C03576=1018.890,246.448,-130.544,169.177,50.795,159.695
C03577=1018.883,246.200,-130.516,169.173,50.800,159.695
C03578=1018.878,245.952,-130.488,169.170,50.806,159.696
C03579=1018.872,245.703,-130.460,169.165,50.812,159.696
C03580=1018.866,245.455,-130.433,169.160,50.817,159.697
C03581=1018.860,245.206,-130.405,169.156,50.823,159.697
C03582=1018.855,244.958,-130.377,169.152,50.829,159.698
C03583=1018.848,244.709,-130.349,169.148,50.834,159.698
C03584=1018.843,244.461,-130.321,169.143,50.840,159.699
C03585=1018.836,244.213,-130.294,169.139,50.846,159.699
C03586=1018.831,243.964,-130.266,169.135,50.852,159.700
C03587=1018.825,243.715,-130.238,169.131,50.857,159.700
C03588=1018.819,243.468,-130.211,169.126,50.863,159.701
C03589=1018.813,243.219,-130.182,169.122,50.869,159.701
C03590=1018.807,242.971,-130.156,169.118,50.875,159.702
C03591=1018.802,242.723,-130.128,169.113,50.881,159.702
C03592=1018.795,242.473,-130.101,169.109,50.887,159.703
C03593=1018.789,242.226,-130.073,169.104,50.893,159.703
C03594=1018.784,241.976,-130.046,169.101,50.899,159.704
C03595=1018.778,241.729,-130.018,169.095,50.904,159.704
C03596=1018.771,241.480,-129.991,169.092,50.910,159.705
C03597=1018.766,241.232,-129.963,169.088,50.917,159.706
C03598=1018.760,240.983,-129.937,169.083,50.922,159.706
C03599=1018.753,240.735,-129.909,169.079,50.928,159.707
C03600=1018.748,240.486,-129.882,169.074,50.934,159.707
C03601=1018.742,240.238,-129.854,169.071,50.940,159.708
C03602=1018.736,239.989,-129.827,169.067,50.946,159.709
C03603=1018.731,239.741,-129.799,169.062,50.952,159.709
C03604=1018.724,239.492,-129.772,169.058,50.958,159.710
C03605=1018.718,239.244,-129.745,169.053,50.965,159.710
C03606=1018.713,238.996,-129.718,169.049,50.970,159.711
C03607=1018.707,238.747,-129.691,169.045,50.976,159.711
C03608=1018.701,238.499,-129.663,169.041,50.983,159.712
C03609=1018.694,238.250,-129.636,169.036,50.989,159.712
C03610=1018.688,238.002,-129.610,169.033,50.995,159.713
C03611=1018.683,237.753,-129.583,169.028,51.001,159.714
C03612=1018.676,237.505,-129.555,169.024,51.007,159.714
C03613=1018.670,237.256,-129.529,169.019,51.013,159.715
C03614=1018.664,237.008,-129.502,169.016,51.020,159.715
C03615=1018.658,236.759,-129.475,169.011,51.026,159.716
C03616=1018.652,236.511,-129.448,169.007,51.032,159.717
C03617=1018.646,236.263,-129.421,169.004,51.038,159.717
C03618=1018.641,236.013,-129.393,168.999,51.045,159.718
C03619=1018.635,235.765,-129.367,168.994,51.051,159.719
C03620=1018.629,235.517,-129.340,168.991,51.057,159.719
C03621=1018.623,235.268,-129.313,168.985,51.063,159.720
C03622=1018.617,235.019,-129.286,168.982,51.069,159.720
C03623=1018.611,234.792,-129.262,168.978,51.075,159.721
C03624=1018.605,234.565,-129.237,168.974,51.081,159.721
C03625=1018.600,234.338,-129.213,168.970,51.087,159.722
C03626=1018.595,234.111,-129.189,168.966,51.092,159.723
C03627=1018.590,233.885,-129.164,168.963,51.098,159.723
C03628=1018.584,233.657,-129.140,168.959,51.104,159.724
C03629=1018.578,233.430,-129.115,168.955,51.110,159.724
C03630=1018.573,233.203,-129.090,168.951,51.116,159.725
C03631=1018.567,232.954,-129.064,168.948,51.122,159.726
C03632=1018.562,232.706,-129.037,168.943,51.129,159.726
C03633=1018.555,232.457,-129.010,168.939,51.135,159.727
C03634=1018.550,232.209,-128.983,168.935,51.141,159.728
C03635=1018.544,231.960,-128.957,168.931,51.147,159.728
C03636=1018.538,231.712,-128.930,168.926,51.154,159.729
C03637=1018.532,231.464,-128.903,168.922,51.160,159.729
C03638=1018.526,231.214,-128.877,168.918,51.166,159.730
C03639=1018.520,230.966,-128.850,168.913,51.173,159.731
C03640=1018.515,230.717,-128.824,168.910,51.180,159.731
C03641=1018.509,230.469,-128.797,168.906,51.186,159.732
C03642=1018.503,230.220,-128.770,168.902,51.192,159.733
C03643=1018.497,229.972,-128.744,168.897,51.199,159.733
C03644=1018.490,229.723,-128.717,168.894,51.205,159.734
C03645=1018.484,229.475,-128.691,168.889,51.212,159.735
C03646=1018.479,229.226,-128.665,168.885,51.218,159.735
C03647=1018.473,228.978,-128.638,168.881,51.225,159.736
C03648=1018.467,228.729,-128.611,168.877,51.232,159.737
C03649=1018.462,228.481,-128.585,168.873,51.238,159.737
C03650=1018.455,228.233,-128.559,168.868,51.244,159.738
C03651=1018.450,227.984,-128.533,168.864,51.252,159.739
C03652=1018.443,227.735,-128.506,168.861,51.258,159.739
C03653=1018.437,227.486,-128.479,168.856,51.264,159.740
C03654=1018.432,227.238,-128.453,168.853,51.271,159.741
C03655=1018.426,226.989,-128.427,168.848,51.278,159.742
C03656=1018.420,226.741,-128.401,168.843,51.284,159.742
C03657=1018.414,226.493,-128.374,168.840,51.291,159.743
C03658=1018.409,226.244,-128.348,168.836,51.297,159.744
C03659=1018.402,225.996,-128.322,168.832,51.304,159.744
C03660=1018.397,225.747,-128.296,168.828,51.311,159.745
C03661=1018.391,225.498,-128.269,168.823,51.318,159.746
C03662=1018.385,225.250,-128.244,168.819,51.324,159.746
C03663=1018.379,225.001,-128.217,168.816,51.331,159.747
C03664=1018.372,224.752,-128.192,168.811,51.338,159.748
C03665=1018.366,224.504,-128.165,168.807,51.345,159.749
C03666=1018.360,224.255,-128.140,168.804,51.352,159.749
C03667=1018.354,224.007,-128.113,168.799,51.358,159.750
C03668=1018.349,223.758,-128.087,168.795,51.365,159.751
C03669=1018.342,223.510,-128.061,168.791,51.372,159.752
C03670=1018.337,223.261,-128.035,168.787,51.379,159.752
C03671=1018.330,223.013,-128.009,168.783,51.386,159.753
C03672=1018.325,222.764,-127.983,168.779,51.393,159.754
C03673=1018.319,222.515,-127.957,168.775,51.399,159.755
C03674=1018.313,222.267,-127.931,168.770,51.406,159.755
C03675=1018.307,222.018,-127.905,168.766,51.414,159.756
C03676=1018.301,221.769,-127.879,168.763,51.420,159.757
C03677=1018.295,221.521,-127.853,168.758,51.427,159.758
C03678=1018.289,221.272,-127.828,168.754,51.434,159.758
C03679=1018.283,221.023,-127.801,168.751,51.440,159.759
C03680=1018.278,220.774,-127.775,168.746,51.448,159.760
C03681=1018.272,220.526,-127.750,168.742,51.455,159.761
C03682=1018.266,220.277,-127.723,168.738,51.462,159.761
C03683=1018.261,220.047,-127.699,168.734,51.468,159.762
C03684=1018.255,219.815,-127.676,168.731,51.474,159.763
C03685=1018.250,219.583,-127.651,168.728,51.481,159.764
C03686=1018.244,219.353,-127.628,168.723,51.488,159.764
C03687=1018.239,219.122,-127.603,168.719,51.494,159.765
C03688=1018.234,218.890,-127.579,168.716,51.501,159.766
C03689=1018.228,218.659,-127.556,168.713,51.507,159.766
C03690=1018.222,218.428,-127.531,168.708,51.513,159.767
C03691=1018.217,218.179,-127.505,168.705,51.520,159.768
C03692=1018.211,217.930,-127.480,168.701,51.527,159.769
C03693=1018.205,217.682,-127.455,168.696,51.535,159.769
C03694=1018.200,217.433,-127.429,168.692,51.542,159.770
C03695=1018.193,217.185,-127.403,168.688,51.549,159.771
C03696=1018.187,216.936,-127.378,168.685,51.556,159.772
C03697=1018.181,216.687,-127.352,168.681,51.563,159.773
C03698=1018.175,216.439,-127.327,168.676,51.570,159.773
C03699=1018.169,216.190,-127.301,168.672,51.578,159.774
C03700=1018.163,215.941,-127.276,168.668,51.585,159.775
C03701=1018.158,215.693,-127.250,168.664,51.592,159.776
C03702=1018.152,215.444,-127.225,168.661,51.599,159.777
C03703=1018.146,215.196,-127.200,168.657,51.607,159.778
C03704=1018.140,214.947,-127.174,168.653,51.614,159.778
C03705=1018.134,214.698,-127.148,168.648,51.621,159.779
C03706=1018.128,214.450,-127.123,168.644,51.629,159.780
C03707=1018.122,214.202,-127.098,168.640,51.636,159.781
C03708=1018.117,213.953,-127.072,168.637,51.643,159.782
C03709=1018.110,213.704,-127.047,168.633,51.650,159.782
C03710=1018.104,213.455,-127.021,168.629,51.658,159.783
C03711=1018.098,213.207,-126.996,168.625,51.665,159.784
C03712=1018.093,212.958,-126.971,168.621,51.672,159.785
C03713=1018.087,212.709,-126.946,168.616,51.680,159.786
C03714=1018.081,212.460,-126.921,168.612,51.687,159.787
C03715=1018.076,212.211,-126.895,168.609,51.694,159.787
C03716=1018.069,211.963,-126.869,168.605,51.702,159.788
C03717=1018.064,211.715,-126.844,168.601,51.709,159.789
C03718=1018.058,211.466,-126.819,168.597,51.716,159.790
C03719=1018.052,211.217,-126.793,168.593,51.723,159.791
C03720=1018.046,210.968,-126.768,168.589,51.731,159.792
C03721=1018.041,210.720,-126.743,168.585,51.739,159.793
C03722=1018.034,210.471,-126.718,168.581,51.746,159.793
C03723=1018.029,210.222,-126.692,168.578,51.753,159.794
C03724=1018.023,209.974,-126.667,168.574,51.761,159.795
C03725=1018.017,209.726,-126.642,168.570,51.768,159.796
C03726=1018.011,209.476,-126.617,168.566,51.776,159.797
C03727=1018.006,209.228,-126.592,168.562,51.783,159.798
C03728=1017.999,208.980,-126.567,168.557,51.790,159.799
C03729=1017.993,208.730,-126.542,168.554,51.798,159.800
C03730=1017.988,208.481,-126.516,168.550,51.806,159.800
C03731=1017.982,208.233,-126.491,168.546,51.813,159.801
C03732=1017.976,207.984,-126.467,168.542,51.821,159.802
C03733=1017.970,207.735,-126.441,168.538,51.829,159.803
C03734=1017.965,207.487,-126.417,168.534,51.836,159.804
C03735=1017.959,207.238,-126.392,168.530,51.844,159.805
C03736=1017.953,206.989,-126.367,168.526,51.851,159.806
C03737=1017.947,206.741,-126.342,168.522,51.859,159.807
C03738=1017.941,206.492,-126.317,168.518,51.866,159.807
C03739=1017.935,206.244,-126.292,168.514,51.874,159.808
C03740=1017.930,205.995,-126.267,168.511,51.882,159.809
C03741=1017.923,205.746,-126.242,168.506,51.890,159.810
C03742=1017.918,205.498,-126.218,168.503,51.898,159.811
C03743=1017.912,205.264,-126.195,168.500,51.904,159.812
C03744=1017.907,205.031,-126.171,168.495,51.912,159.813
C03745=1017.901,204.798,-126.148,168.491,51.919,159.814
C03746=1017.895,204.565,-126.125,168.489,51.927,159.815
C03747=1017.890,204.332,-126.102,168.484,51.934,159.816
C03748=1017.885,204.098,-126.078,168.481,51.941,159.816
C03749=1017.879,203.865,-126.055,168.478,51.949,159.817
C03750=1017.854,202.631,-125.940,167.998,51.859,159.707
C03751=1017.849,202.382,-125.916,167.994,51.868,159.708
C03752=1017.844,202.134,-125.893,167.989,51.876,159.709
C03753=1017.839,201.884,-125.870,167.984,51.885,159.710
C03754=1017.834,201.636,-125.847,167.980,51.894,159.711
C03755=1017.828,201.387,-125.824,167.976,51.903,159.712
C03756=1017.824,201.138,-125.801,167.971,51.912,159.713
C03757=1017.819,200.889,-125.778,167.966,51.921,159.714
C03758=1017.815,200.640,-125.755,167.962,51.930,159.715
C03759=1017.809,200.391,-125.732,167.956,51.938,159.716
C03760=1017.805,200.143,-125.709,167.952,51.947,159.717
C03761=1017.800,199.893,-125.686,167.948,51.956,159.718
C03762=1017.795,199.645,-125.663,167.943,51.965,159.719
C03763=1017.790,199.395,-125.640,167.938,51.974,159.720
C03764=1017.785,199.147,-125.617,167.934,51.983,159.721
C03765=1017.780,198.897,-125.594,167.930,51.992,159.722
C03766=1017.775,198.649,-125.572,167.925,52.001,159.723
C03767=1017.770,198.400,-125.549,167.921,52.010,159.724
C03768=1017.765,198.151,-125.526,167.916,52.019,159.725
C03769=1017.760,197.902,-125.504,167.912,52.028,159.726
C03770=1017.755,197.654,-125.481,167.907,52.037,159.727
C03771=1017.750,197.404,-125.459,167.903,52.046,159.728
C03772=1017.745,197.156,-125.436,167.898,52.055,159.729
C03773=1017.739,196.906,-125.414,167.893,52.064,159.730
C03774=1017.735,196.657,-125.391,167.889,52.073,159.731
C03775=1017.730,196.408,-125.368,167.885,52.082,159.732
C03776=1017.725,196.159,-125.346,167.880,52.091,159.733
C03777=1017.720,195.911,-125.323,167.875,52.100,159.734
C03778=1017.715,195.661,-125.301,167.871,52.109,159.735
C03779=1017.710,195.413,-125.278,167.867,52.118,159.736
C03780=1017.704,195.163,-125.256,167.862,52.127,159.737
C03781=1017.700,194.915,-125.233,167.858,52.136,159.738
C03782=1017.695,194.666,-125.211,167.854,52.145,159.739
C03783=1017.690,194.417,-125.189,167.849,52.154,159.740
C03784=1017.685,194.168,-125.166,167.845,52.163,159.741
C03785=1017.681,193.919,-125.144,167.841,52.173,159.742
C03786=1017.675,193.670,-125.122,167.836,52.182,159.743
C03787=1017.671,193.421,-125.099,167.832,52.191,159.744
C03788=1017.666,193.172,-125.077,167.827,52.199,159.745
C03789=1017.661,192.923,-125.054,167.823,52.208,159.746
C03790=1017.656,192.674,-125.031,167.819,52.217,159.747
C03791=1017.651,192.426,-125.009,167.814,52.226,159.748
C03792=1017.646,192.176,-124.987,167.810,52.236,159.749
C03793=1017.641,191.927,-124.965,167.806,52.245,159.750
C03794=1017.637,191.679,-124.942,167.801,52.254,159.751
C03795=1017.631,191.429,-124.920,167.797,52.263,159.752
C03796=1017.626,191.180,-124.898,167.793,52.272,159.753
C03797=1017.622,190.931,-124.876,167.788,52.281,159.754
C03798=1017.617,190.683,-124.853,167.784,52.290,159.755
C03799=1017.612,190.434,-124.831,167.780,52.299,159.756
C03800=1017.607,190.185,-124.809,167.775,52.308,159.757
C03801=1017.603,189.936,-124.786,167.771,52.317,159.758
C03802=1017.598,189.687,-124.765,167.766,52.326,159.759
C03803=1017.592,189.438,-124.742,167.762,52.335,159.760
C03804=1017.588,189.189,-124.719,167.758,52.344,159.761
C03805=1017.583,188.940,-124.697,167.754,52.353,159.762
C03806=1017.579,188.691,-124.675,167.750,52.362,159.764
C03807=1017.574,188.441,-124.653,167.746,52.371,159.765
C03808=1017.569,188.193,-124.631,167.742,52.381,159.766
C03809=1017.564,187.944,-124.609,167.737,52.390,159.767
C03810=1017.559,187.696,-124.586,167.733,52.399,159.768
C03811=1017.554,187.415,-124.561,167.728,52.409,159.769
C03812=1017.548,187.135,-124.536,167.723,52.419,159.770
C03813=1017.544,186.854,-124.511,167.719,52.429,159.771
C03814=1017.538,186.573,-124.486,167.714,52.440,159.772
C03815=1017.534,186.324,-124.464,167.710,52.448,159.773
C03816=1017.529,186.076,-124.442,167.706,52.458,159.774
C03817=1017.524,185.826,-124.420,167.702,52.467,159.775
C03818=1017.519,185.577,-124.398,167.698,52.476,159.777
C03819=1017.515,185.328,-124.375,167.693,52.485,159.778
C03820=1017.510,185.079,-124.354,167.689,52.493,159.778
C03821=1017.505,184.830,-124.332,167.685,52.502,159.780
C03822=1017.500,184.582,-124.310,167.681,52.511,159.781
C03823=1017.496,184.333,-124.287,167.677,52.521,159.782
C03824=1017.491,184.084,-124.266,167.673,52.530,159.783
C03825=1017.486,183.835,-124.244,167.668,52.539,159.784
C03826=1017.482,183.586,-124.221,167.664,52.548,159.785
C03827=1017.477,183.336,-124.199,167.661,52.557,159.786
C03828=1017.472,183.087,-124.178,167.657,52.566,159.787
C03829=1017.468,182.838,-124.156,167.652,52.575,159.788
C03830=1017.463,182.589,-124.134,167.648,52.584,159.789
C03831=1017.459,182.340,-124.112,167.644,52.594,159.790
C03832=1017.454,182.091,-124.090,167.641,52.602,159.791
C03833=1017.450,181.842,-124.067,167.636,52.611,159.792
C03834=1017.444,181.593,-124.047,167.632,52.621,159.793
C03835=1017.440,181.344,-124.025,167.628,52.630,159.794
C03836=1017.435,181.095,-124.004,167.624,52.639,159.795
C03837=1017.429,180.846,-123.982,167.619,52.648,159.796
C03838=1017.424,180.597,-123.960,167.616,52.658,159.798
C03839=1017.419,180.348,-123.940,167.611,52.667,159.799
C03840=1017.414,180.099,-123.918,167.607,52.677,159.800
C03841=1017.410,179.849,-123.897,167.603,52.687,159.801
C03842=1017.404,179.601,-123.875,167.599,52.696,159.802
C03843=1017.399,179.351,-123.854,167.595,52.705,159.803
C03844=1017.395,179.103,-123.832,167.591,52.714,159.804
C03845=1017.389,178.853,-123.812,167.587,52.724,159.805
C03846=1017.385,178.605,-123.790,167.583,52.733,159.806
C03847=1017.380,178.355,-123.769,167.579,52.742,159.808
C03848=1017.374,178.107,-123.748,167.575,52.751,159.809
C03849=1017.370,177.857,-123.726,167.571,52.761,159.810
C03850=1017.365,177.608,-123.706,167.567,52.770,159.811
C03851=1017.360,177.359,-123.684,167.563,52.780,159.812
C03852=1017.355,177.110,-123.663,167.559,52.789,159.813
C03853=1017.350,176.861,-123.642,167.555,52.799,159.814
C03854=1017.345,176.612,-123.620,167.551,52.808,159.815
C03855=1017.341,176.363,-123.599,167.547,52.817,159.816
C03856=1017.335,176.114,-123.578,167.542,52.827,159.817
C03857=1017.331,175.865,-123.557,167.540,52.836,159.819
C03858=1017.325,175.616,-123.536,167.535,52.845,159.820
C03859=1017.321,175.367,-123.515,167.531,52.855,159.821
C03860=1017.316,175.117,-123.493,167.527,52.864,159.822
C03861=1017.311,174.869,-123.472,167.523,52.874,159.823
C03862=1017.306,174.619,-123.451,167.519,52.883,159.824
C03863=1017.301,174.371,-123.431,167.515,52.892,159.825
C03864=1017.297,174.122,-123.409,167.511,52.901,159.826
C03865=1017.292,173.873,-123.388,167.508,52.911,159.828
C03866=1017.287,173.623,-123.367,167.504,52.920,159.829
C03867=1017.282,173.375,-123.345,167.500,52.929,159.830
C03868=1017.277,173.125,-123.324,167.495,52.939,159.831
C03869=1017.272,172.876,-123.304,167.492,52.949,159.832
C03870=1017.268,172.627,-123.282,167.489,52.958,159.833
C03871=1017.262,172.378,-123.261,167.484,52.967,159.834
C03872=1017.258,172.129,-123.240,167.480,52.976,159.835
C03873=1017.254,171.880,-123.219,167.477,52.986,159.837
C03874=1017.248,171.631,-123.199,167.472,52.995,159.838
C03875=1017.243,171.350,-123.174,167.468,53.006,159.839
C03876=1017.238,171.069,-123.151,167.464,53.016,159.840
C03877=1017.232,170.788,-123.127,167.460,53.027,159.841
C03878=1017.227,170.508,-123.104,167.455,53.037,159.842
C03879=1017.222,170.259,-123.083,167.451,53.047,159.844
C03880=1017.218,170.009,-123.061,167.448,53.056,159.845
C03881=1017.212,169.760,-123.041,167.444,53.065,159.846
C03882=1017.208,169.511,-123.020,167.440,53.074,159.847
C03883=1017.203,169.263,-122.999,167.436,53.084,159.848
C03884=1017.198,169.013,-122.978,167.433,53.093,159.849
C03885=1017.194,168.764,-122.957,167.429,53.103,159.850
C03886=1017.189,168.515,-122.936,167.425,53.112,159.851
C03887=1017.184,168.265,-122.915,167.421,53.122,159.853
C03888=1017.180,168.017,-122.895,167.418,53.131,159.854
C03889=1017.175,167.767,-122.874,167.414,53.140,159.855
C03890=1017.170,167.518,-122.852,167.410,53.149,159.856
C03891=1017.165,167.270,-122.831,167.405,53.159,159.857
C03892=1017.161,167.021,-122.810,167.403,53.168,159.858
C03893=1017.156,166.772,-122.790,167.399,53.177,159.860
C03894=1017.151,166.522,-122.769,167.395,53.187,159.861
C03895=1017.147,166.273,-122.747,167.391,53.196,159.862
C03896=1017.142,166.024,-122.727,167.387,53.205,159.863
C03897=1017.138,165.775,-122.706,167.384,53.215,159.864
C03898=1017.132,165.526,-122.686,167.381,53.224,159.865
C03899=1017.128,165.277,-122.665,167.376,53.233,159.866
C03900=1017.124,165.028,-122.644,167.372,53.243,159.867
C03901=1017.119,164.779,-122.623,167.370,53.252,159.869
C03902=1017.114,164.529,-122.602,167.366,53.261,159.870
C03903=1017.109,164.281,-122.582,167.361,53.271,159.871
C03904=1017.105,164.031,-122.561,167.358,53.280,159.872
C03905=1017.100,163.782,-122.539,167.354,53.289,159.873
C03906=1017.096,163.533,-122.519,167.350,53.298,159.874
C03907=1017.091,163.284,-122.498,167.348,53.308,159.875
C03908=1017.086,163.035,-122.478,167.343,53.317,159.876
C03909=1017.082,162.786,-122.457,167.339,53.327,159.878
C03910=1017.078,162.537,-122.436,167.336,53.336,159.879
C03911=1017.073,162.288,-122.415,167.332,53.345,159.880
C03912=1017.068,162.039,-122.394,167.329,53.355,159.881
C03913=1017.063,161.789,-122.374,167.325,53.364,159.882
C03914=1017.059,161.540,-122.354,167.321,53.373,159.883
C03915=1017.054,161.291,-122.333,167.318,53.382,159.884
C03916=1017.050,161.042,-122.312,167.314,53.392,159.885
C03917=1017.046,160.793,-122.291,167.310,53.401,159.886
C03918=1017.041,160.544,-122.271,167.308,53.411,159.888
C03919=1017.037,160.295,-122.250,167.303,53.420,159.889
C03920=1017.031,160.046,-122.229,167.300,53.429,159.890
C03921=1017.027,159.796,-122.209,167.296,53.438,159.891
C03922=1017.023,159.547,-122.188,167.292,53.448,159.892
C03923=1017.018,159.298,-122.168,167.289,53.456,159.893
C03924=1017.014,159.049,-122.147,167.286,53.467,159.895
C03925=1017.009,158.800,-122.126,167.283,53.475,159.896
C03926=1017.005,158.552,-122.105,167.278,53.485,159.897
C03927=1017.000,158.302,-122.086,167.275,53.494,159.898
C03928=1016.995,158.053,-122.065,167.272,53.504,159.899
C03929=1016.990,157.804,-122.046,167.268,53.513,159.900
C03930=1016.985,157.555,-122.025,167.264,53.523,159.901
C03931=1016.981,157.305,-122.005,167.261,53.532,159.903
C03932=1016.976,157.056,-121.984,167.257,53.542,159.904
C03933=1016.972,156.808,-121.964,167.254,53.552,159.905
C03934=1016.967,156.558,-121.944,167.250,53.561,159.906
C03935=1016.961,156.309,-121.924,167.246,53.570,159.907
C03936=1016.957,156.060,-121.904,167.243,53.580,159.909
C03937=1016.952,155.811,-121.884,167.239,53.590,159.910
C03938=1016.947,155.562,-121.864,167.236,53.599,159.911
C03939=1016.942,155.280,-121.841,167.232,53.610,159.912
C03940=1016.937,154.999,-121.819,167.229,53.620,159.914
C03941=1016.931,154.718,-121.796,167.224,53.631,159.915
C03942=1016.926,154.437,-121.774,167.220,53.642,159.916
C03943=1016.922,154.187,-121.753,167.217,53.651,159.917
C03944=1016.917,153.939,-121.733,167.213,53.661,159.919
C03945=1016.912,153.689,-121.713,167.209,53.671,159.920
C03946=1016.908,153.441,-121.693,167.206,53.680,159.921
C03947=1016.903,153.191,-121.673,167.203,53.690,159.922
C03948=1016.897,152.942,-121.653,167.199,53.699,159.923
C03949=1016.893,152.693,-121.633,167.196,53.709,159.925
C03950=1016.888,152.443,-121.613,167.192,53.718,159.926
C03951=1016.883,152.195,-121.593,167.188,53.728,159.927
C03952=1016.879,151.946,-121.574,167.186,53.737,159.928
C03953=1016.874,151.696,-121.554,167.182,53.747,159.929
C03954=1016.870,151.448,-121.534,167.178,53.757,159.931
C03955=1016.865,151.198,-121.514,167.175,53.766,159.932
C03956=1016.860,150.949,-121.494,167.172,53.776,159.933
C03957=1016.855,150.699,-121.475,167.168,53.785,159.934
C03958=1016.851,150.451,-121.454,167.165,53.795,159.936
C03959=1016.846,150.201,-121.435,167.161,53.804,159.937
C03960=1016.841,149.952,-121.415,167.158,53.814,159.938
C03961=1016.836,149.702,-121.395,167.155,53.824,159.939
C03962=1016.832,149.454,-121.375,167.151,53.833,159.940
C03963=1016.827,149.205,-121.356,167.148,53.843,159.941
C03964=1016.822,148.955,-121.336,167.144,53.852,159.943
C03965=1016.817,148.706,-121.317,167.140,53.862,159.944
C03966=1016.812,148.457,-121.296,167.138,53.871,159.945
C03967=1016.808,148.208,-121.277,167.134,53.881,159.946
C03968=1016.803,147.959,-121.257,167.131,53.891,159.947
C03969=1016.798,147.709,-121.238,167.127,53.900,159.949
C03970=1016.794,147.460,-121.218,167.123,53.909,159.950
C03971=1016.789,147.211,-121.198,167.121,53.919,159.951
C03972=1016.784,146.962,-121.178,167.117,53.929,159.952
C03973=1016.780,146.713,-121.159,167.114,53.938,159.953
C03974=1016.775,146.463,-121.139,167.110,53.948,159.955
C03975=1016.770,146.214,-121.120,167.107,53.958,159.956
C03976=1016.766,145.965,-121.100,167.104,53.967,159.957
C03977=1016.761,145.716,-121.081,167.100,53.976,159.958
C03978=1016.756,145.467,-121.061,167.096,53.987,159.959
C03979=1016.752,145.218,-121.042,167.093,53.996,159.961
C03980=1016.746,144.968,-121.022,167.090,54.006,159.962
C03981=1016.742,144.719,-121.003,167.087,54.015,159.963
C03982=1016.737,144.469,-120.983,167.084,54.025,159.964
C03983=1016.732,144.221,-120.964,167.080,54.034,159.965
C03984=1016.728,143.972,-120.945,167.077,54.044,159.967
C03985=1016.723,143.722,-120.925,167.073,54.054,159.968
C03986=1016.718,143.473,-120.906,167.070,54.064,159.969
C03987=1016.713,143.224,-120.887,167.067,54.073,159.970
C03988=1016.708,142.974,-120.867,167.063,54.083,159.972
C03989=1016.703,142.726,-120.848,167.061,54.092,159.973
C03990=1016.699,142.477,-120.828,167.057,54.102,159.974
C03991=1016.695,142.228,-120.809,167.053,54.112,159.975
C03992=1016.689,141.978,-120.790,167.051,54.122,159.977
C03993=1016.685,141.729,-120.770,167.047,54.131,159.978
C03994=1016.680,141.479,-120.751,167.043,54.141,159.979
C03995=1016.675,141.230,-120.732,167.040,54.150,159.980
C03996=1016.670,140.981,-120.713,167.037,54.161,159.981
C03997=1016.666,140.732,-120.693,167.034,54.170,159.983
C03998=1016.661,140.483,-120.674,167.031,54.180,159.984
C03999=1016.656,140.233,-120.655,167.028,54.189,159.985
C04000=1016.652,139.984,-120.635,167.024,54.199,159.986
C04001=1016.647,139.735,-120.617,167.020,54.209,159.987
C04002=1016.643,139.486,-120.597,167.018,54.218,159.989
C04003=1016.637,139.204,-120.575,167.014,54.229,159.990
C04004=1016.632,138.923,-120.553,167.011,54.240,159.992
C04005=1016.626,138.642,-120.533,167.006,54.250,159.993
C04006=1016.621,138.361,-120.511,167.003,54.261,159.994
C04007=1016.616,138.112,-120.491,167.000,54.272,159.996
C04008=1016.612,137.863,-120.471,166.997,54.281,159.997
C04009=1016.607,137.613,-120.453,166.993,54.290,159.998
C04010=1016.603,137.364,-120.434,166.991,54.300,159.999
C04011=1016.597,137.115,-120.414,166.987,54.310,160.001
C04012=1016.593,136.865,-120.396,166.983,54.320,160.002
C04013=1016.588,136.616,-120.377,166.981,54.330,160.003
C04014=1016.584,136.367,-120.357,166.977,54.339,160.004
C04015=1016.579,136.118,-120.339,166.975,54.349,160.006
C04016=1016.574,135.868,-120.319,166.971,54.358,160.007
C04017=1016.569,135.619,-120.300,166.968,54.369,160.008
C04018=1016.565,135.370,-120.282,166.965,54.378,160.009
C04019=1016.560,135.121,-120.263,166.961,54.388,160.011
C04020=1016.555,134.872,-120.244,166.958,54.397,160.012
C04021=1016.550,134.622,-120.225,166.955,54.407,160.013
C04022=1016.545,134.373,-120.206,166.952,54.416,160.014
C04023=1016.541,134.124,-120.187,166.949,54.427,160.016
C04024=1016.536,133.875,-120.168,166.945,54.436,160.017
C04025=1016.531,133.626,-120.150,166.943,54.446,160.018
C04026=1016.527,133.376,-120.131,166.939,54.456,160.019
C04027=1016.521,133.127,-120.111,166.936,54.465,160.021
C04028=1016.517,132.877,-120.093,166.933,54.475,160.022
C04029=1016.512,132.629,-120.074,166.930,54.485,160.023
C04030=1016.507,132.379,-120.056,166.926,54.494,160.024
C04031=1016.503,132.130,-120.036,166.924,54.504,160.026
C04032=1016.498,131.881,-120.018,166.920,54.514,160.027
C04033=1016.494,131.632,-119.999,166.917,54.524,160.028
C04034=1016.489,131.383,-119.980,166.914,54.533,160.029
C04035=1016.483,131.133,-119.961,166.911,54.543,160.030
C04036=1016.479,130.883,-119.942,166.908,54.553,160.032
C04037=1016.474,130.635,-119.923,166.905,54.563,160.033
C04038=1016.469,130.385,-119.905,166.902,54.572,160.034
C04039=1016.465,130.136,-119.887,166.898,54.582,160.035
C04040=1016.460,129.887,-119.868,166.896,54.591,160.037
C04041=1016.456,129.637,-119.849,166.892,54.601,160.038
C04042=1016.451,129.389,-119.830,166.890,54.611,160.039
C04043=1016.446,129.138,-119.812,166.886,54.621,160.041
C04044=1016.441,128.889,-119.793,166.883,54.630,160.042
C04045=1016.436,128.640,-119.775,166.880,54.641,160.043
C04046=1016.431,128.391,-119.756,166.877,54.651,160.044
C04047=1016.426,128.142,-119.738,166.874,54.660,160.046
C04048=1016.421,127.892,-119.720,166.871,54.670,160.047
C04049=1016.417,127.643,-119.702,166.867,54.681,160.048
C04050=1016.412,127.394,-119.683,166.865,54.690,160.049
C04051=1016.407,127.145,-119.665,166.861,54.700,160.051
C04052=1016.402,126.896,-119.647,166.858,54.709,160.052
C04053=1016.397,126.646,-119.628,166.855,54.719,160.053
C04054=1016.392,126.397,-119.610,166.852,54.730,160.055
C04055=1016.388,126.148,-119.591,166.849,54.739,160.056
C04056=1016.383,125.898,-119.573,166.846,54.749,160.057
C04057=1016.379,125.649,-119.555,166.844,54.759,160.059
C04058=1016.373,125.399,-119.536,166.840,54.769,160.060
C04059=1016.368,125.150,-119.518,166.836,54.779,160.061
C04060=1016.364,124.900,-119.500,166.834,54.788,160.062
C04061=1016.358,124.652,-119.481,166.830,54.799,160.063
C04062=1016.354,124.402,-119.463,166.828,54.808,160.065
C04063=1016.349,124.153,-119.444,166.824,54.818,160.066
C04064=1016.344,123.904,-119.426,166.822,54.828,160.068
C04065=1016.339,123.654,-119.408,166.818,54.838,160.069
C04066=1016.335,123.405,-119.390,166.816,54.847,160.070
C04067=1016.329,123.124,-119.369,166.812,54.859,160.071
C04068=1016.324,122.843,-119.349,166.809,54.869,160.073
C04069=1016.319,122.562,-119.328,166.805,54.881,160.074
C04070=1016.313,122.281,-119.308,166.803,54.892,160.076
C04071=1016.308,122.031,-119.290,166.799,54.901,160.077
C04072=1016.304,121.782,-119.272,166.797,54.911,160.078
C04073=1016.299,121.533,-119.253,166.793,54.921,160.079
C04074=1016.294,121.283,-119.235,166.791,54.931,160.081
C04075=1016.289,121.034,-119.217,166.787,54.940,160.082
C04076=1016.285,120.785,-119.199,166.785,54.950,160.083
C04077=1016.280,120.535,-119.181,166.781,54.960,160.084
C04078=1016.275,120.286,-119.163,166.779,54.970,160.086
C04079=1016.270,120.037,-119.144,166.775,54.979,160.087
C04080=1016.265,119.787,-119.126,166.773,54.989,160.089
C04081=1016.261,119.538,-119.108,166.769,54.999,160.090
C04082=1016.256,119.289,-119.090,166.767,55.009,160.091
C04083=1016.251,119.039,-119.072,166.763,55.019,160.092
C04084=1016.247,118.790,-119.052,166.761,55.028,160.094
C04085=1016.243,118.542,-119.034,166.757,55.038,160.095
C04086=1016.238,118.292,-119.017,166.755,55.048,160.096
C04087=1016.233,118.042,-118.999,166.751,55.058,160.097
C04088=1016.228,117.793,-118.981,166.749,55.068,160.099
C04089=1016.224,117.544,-118.963,166.745,55.077,160.100
C04090=1016.219,117.294,-118.944,166.743,55.087,160.101
C04091=1016.214,117.045,-118.926,166.739,55.097,160.102
C04092=1016.209,116.795,-118.908,166.737,55.106,160.104
C04093=1016.205,116.546,-118.890,166.735,55.116,160.105
C04094=1016.200,116.297,-118.872,166.731,55.126,160.106
C04095=1016.196,116.048,-118.854,166.729,55.136,160.108
C04096=1016.191,115.799,-118.836,166.725,55.145,160.109
C04097=1016.186,115.549,-118.818,166.723,55.155,160.110
C04098=1016.181,115.300,-118.799,166.720,55.165,160.111
C04099=1016.177,115.051,-118.781,166.716,55.174,160.113
C04100=1016.172,114.801,-118.763,166.714,55.184,160.114
C04101=1016.168,114.553,-118.745,166.711,55.194,160.115
C04102=1016.163,114.303,-118.727,166.708,55.203,160.116
C04103=1016.158,114.053,-118.710,166.706,55.213,160.118
C04104=1016.154,113.804,-118.692,166.702,55.223,160.119
C04105=1016.149,113.555,-118.673,166.700,55.233,160.120
C04106=1016.144,113.305,-118.655,166.696,55.242,160.121
C04107=1016.140,113.057,-118.637,166.694,55.252,160.123
C04108=1016.135,112.807,-118.619,166.692,55.262,160.124
C04109=1016.130,112.558,-118.601,166.688,55.271,160.125
C04110=1016.125,112.309,-118.583,166.685,55.281,160.126
C04111=1016.121,112.059,-118.566,166.683,55.291,160.128
C04112=1016.117,111.810,-118.548,166.679,55.300,160.129
C04113=1016.112,111.561,-118.530,166.677,55.310,160.131
C04114=1016.107,111.311,-118.513,166.674,55.320,160.132
C04115=1016.102,111.062,-118.495,166.672,55.330,160.133
C04116=1016.097,110.812,-118.476,166.668,55.340,160.134
C04117=1016.093,110.563,-118.460,166.666,55.350,160.136
C04118=1016.088,110.314,-118.442,166.662,55.359,160.137
C04119=1016.083,110.065,-118.424,166.660,55.369,160.138
C04120=1016.079,109.815,-118.406,166.656,55.379,160.139
C04121=1016.073,109.566,-118.389,166.654,55.388,160.141
C04122=1016.069,109.317,-118.371,166.652,55.398,160.142
C04123=1016.064,109.067,-118.353,166.648,55.408,160.143
C04124=1016.059,108.818,-118.336,166.646,55.418,160.145
C04125=1016.054,108.568,-118.318,166.643,55.428,160.146
C04126=1016.049,108.320,-118.301,166.640,55.438,160.147
C04127=1016.045,108.070,-118.284,166.637,55.448,160.149
C04128=1016.040,107.821,-118.266,166.634,55.457,160.150
C04129=1016.035,107.571,-118.249,166.631,55.468,160.151
C04130=1016.030,107.322,-118.231,166.629,55.477,160.152
C04131=1016.025,107.041,-118.212,166.625,55.489,160.154
C04132=1016.019,106.759,-118.192,166.623,55.500,160.156
C04133=1016.014,106.479,-118.172,166.618,55.511,160.157
C04134=1016.008,106.197,-118.153,166.616,55.522,160.158
C04135=1016.004,105.948,-118.136,166.613,55.532,160.160
C04136=1015.999,105.699,-118.118,166.610,55.541,160.161
C04137=1015.994,105.449,-118.101,166.607,55.552,160.162
C04138=1015.989,105.200,-118.083,166.604,55.561,160.164
C04139=1015.985,104.950,-118.066,166.602,55.571,160.165
C04140=1015.979,104.701,-118.048,166.599,55.581,160.166
C04141=1015.975,104.451,-118.031,166.596,55.590,160.167
C04142=1015.970,104.202,-118.014,166.593,55.601,160.169
C04143=1015.966,103.953,-117.996,166.591,55.610,160.170
C04144=1015.961,103.703,-117.979,166.587,55.620,160.171
C04145=1015.956,103.454,-117.961,166.585,55.630,160.173
C04146=1015.952,103.205,-117.944,166.583,55.640,160.174
C04147=1015.946,102.956,-117.927,166.579,55.650,160.175
C04148=1015.942,102.706,-117.909,166.577,55.660,160.177
C04149=1015.937,102.457,-117.893,166.574,55.669,160.178
C04150=1015.932,102.207,-117.874,166.571,55.679,160.179
C04151=1015.927,101.958,-117.858,166.569,55.689,160.181
C04152=1015.923,101.709,-117.841,166.566,55.698,160.182
C04153=1015.918,101.460,-117.823,166.564,55.709,160.183
C04154=1015.914,101.210,-117.806,166.560,55.718,160.184
C04155=1015.909,100.961,-117.789,166.557,55.728,160.186
C04156=1015.904,100.711,-117.771,166.555,55.738,160.187
C04157=1015.899,100.462,-117.754,166.552,55.747,160.188
C04158=1015.895,100.212,-117.737,166.549,55.757,160.189
C04159=1015.889,99.963,-117.719,166.547,55.767,160.191
C04160=1015.885,99.714,-117.702,166.544,55.777,160.192
C04161=1015.880,99.464,-117.685,166.541,55.786,160.193
C04162=1015.875,99.215,-117.667,166.538,55.796,160.195
C04163=1015.871,98.966,-117.651,166.536,55.806,160.196
C04164=1015.866,98.716,-117.633,166.534,55.816,160.197
C04165=1015.862,98.467,-117.617,166.530,55.826,160.199
C04166=1015.856,98.217,-117.600,166.528,55.836,160.200
C04167=1015.851,97.968,-117.582,166.525,55.845,160.201
C04168=1015.847,97.719,-117.565,166.523,55.855,160.203
C04169=1015.842,97.469,-117.549,166.519,55.865,160.204
C04170=1015.837,97.221,-117.532,166.517,55.875,160.205
C04171=1015.832,96.971,-117.515,166.514,55.885,160.206
C04172=1015.828,96.721,-117.498,166.511,55.894,160.208
C04173=1015.823,96.472,-117.481,166.509,55.905,160.209
C04174=1015.818,96.222,-117.464,166.506,55.914,160.210
C04175=1015.813,95.973,-117.448,166.504,55.924,160.212
C04176=1015.808,95.724,-117.431,166.500,55.934,160.213
C04177=1015.803,95.474,-117.413,166.498,55.944,160.214
C04178=1015.798,95.225,-117.396,166.495,55.954,160.216
C04179=1015.793,94.976,-117.380,166.492,55.963,160.217
C04180=1015.789,94.727,-117.363,166.490,55.974,160.218
C04181=1015.784,94.477,-117.346,166.487,55.983,160.219
C04182=1015.780,94.228,-117.329,166.485,55.993,160.221
C04183=1015.774,93.978,-117.312,166.481,56.003,160.222
C04184=1015.770,93.729,-117.296,166.479,56.013,160.223
C04185=1015.765,93.480,-117.279,166.477,56.023,160.225
C04186=1015.760,93.230,-117.262,166.473,56.033,160.226
C04187=1015.755,92.981,-117.245,166.471,56.043,160.228
C04188=1015.750,92.731,-117.228,166.469,56.052,160.229
C04189=1015.746,92.482,-117.212,166.465,56.062,160.230
C04190=1015.741,92.232,-117.194,166.464,56.072,160.231
C04191=1015.737,91.983,-117.178,166.460,56.082,160.233
C04192=1015.731,91.733,-117.161,166.458,56.091,160.234
C04193=1015.727,91.484,-117.144,166.456,56.101,160.235
C04194=1015.722,91.235,-117.128,166.452,56.111,160.236
C04195=1015.716,90.893,-117.105,166.449,56.125,160.238
C04196=1015.710,90.552,-117.082,166.445,56.137,160.240
C04197=1015.702,90.210,-117.059,166.441,56.151,160.242
C04198=1015.696,89.869,-117.035,166.438,56.164,160.244
C04199=1015.691,89.620,-117.019,166.436,56.174,160.245
C04200=1015.686,89.371,-117.002,166.433,56.183,160.246
C04201=1015.683,89.121,-116.986,166.430,56.194,160.248
C04202=1015.677,88.871,-116.969,166.428,56.203,160.249
C04203=1015.673,88.622,-116.952,166.425,56.213,160.250
C04204=1015.667,88.373,-116.936,166.422,56.223,160.252
C04205=1015.663,88.124,-116.919,166.420,56.233,160.253
C04206=1015.658,87.873,-116.903,166.417,56.242,160.254
C04207=1015.653,87.624,-116.886,166.415,56.253,160.255
C04208=1015.647,87.375,-116.870,166.411,56.262,160.257
C04209=1015.643,87.126,-116.854,166.409,56.273,160.258
C04210=1015.638,86.876,-116.838,166.407,56.282,160.259
C04211=1015.633,86.627,-116.821,166.404,56.292,160.261
C04212=1015.629,86.378,-116.805,166.402,56.302,160.262
C04213=1015.623,86.128,-116.788,166.398,56.312,160.263
C04214=1015.619,85.879,-116.772,166.396,56.322,160.265
C04215=1015.614,85.629,-116.755,166.394,56.331,160.266
C04216=1015.609,85.380,-116.739,166.391,56.341,160.267
C04217=1015.604,85.131,-116.723,166.389,56.351,160.269
C04218=1015.599,84.881,-116.707,166.385,56.361,160.270
C04219=1015.594,84.632,-116.690,166.383,56.371,160.271
C04220=1015.590,84.382,-116.674,166.381,56.381,160.273
C04221=1015.585,84.133,-116.658,166.378,56.391,160.274
C04222=1015.580,83.883,-116.641,166.375,56.400,160.275
C04223=1015.575,83.634,-116.625,166.373,56.410,160.277
C04224=1015.571,83.385,-116.608,166.370,56.420,160.278
C04225=1015.566,83.135,-116.592,166.368,56.430,160.279
C04226=1015.561,82.885,-116.576,166.365,56.439,160.280
C04227=1015.556,82.637,-116.560,166.362,56.450,160.282
C04228=1015.551,82.386,-116.544,166.360,56.459,160.283
C04229=1015.546,82.138,-116.527,166.358,56.469,160.284
C04230=1015.541,81.888,-116.510,166.354,56.478,160.285
C04231=1015.537,81.638,-116.495,166.353,56.489,160.287
C04232=1015.532,81.389,-116.478,166.350,56.498,160.288
C04233=1015.527,81.139,-116.462,166.347,56.508,160.289
C04234=1015.523,80.890,-116.446,166.344,56.517,160.291
C04235=1015.518,80.641,-116.429,166.343,56.528,160.292
C04236=1015.512,80.391,-116.414,166.339,56.537,160.293
C04237=1015.508,80.142,-116.397,166.337,56.547,160.295
C04238=1015.504,79.893,-116.381,166.335,56.556,160.296
C04239=1015.500,79.673,-116.367,166.332,56.565,160.297
C04240=1015.495,79.454,-116.353,166.330,56.573,160.298
C04241=1015.491,79.235,-116.338,166.328,56.582,160.299
C04242=1015.487,79.016,-116.324,166.325,56.590,160.300
C04243=1015.482,78.797,-116.310,166.323,56.599,160.302
C04244=1015.478,78.577,-116.295,166.321,56.608,160.303
C04245=1015.474,78.358,-116.281,166.319,56.617,160.304
C04246=1015.470,78.139,-116.267,166.317,56.625,160.305
C04247=1015.465,77.889,-116.251,166.314,56.635,160.306
C04248=1015.461,77.640,-116.234,166.312,56.644,160.308
C04249=1015.456,77.390,-116.218,166.309,56.654,160.309
C04250=1015.452,77.141,-116.202,166.307,56.663,160.310
C04251=1015.446,76.892,-116.186,166.304,56.673,160.311
C04252=1015.441,76.643,-116.170,166.301,56.683,160.313
C04253=1015.437,76.393,-116.154,166.300,56.693,160.314
C04254=1015.431,76.144,-116.138,166.296,56.703,160.315
C04255=1015.427,75.894,-116.122,166.294,56.712,160.317
C04256=1015.423,75.644,-116.106,166.292,56.722,160.318
C04257=1015.417,75.395,-116.089,166.288,56.732,160.319
C04258=1015.412,75.146,-116.074,166.287,56.742,160.321
C04259=1015.407,74.864,-116.057,166.284,56.752,160.322
C04260=1015.402,74.584,-116.038,166.281,56.763,160.324
C04261=1015.396,74.303,-116.020,166.278,56.775,160.325
C04262=1015.390,74.022,-116.003,166.275,56.786,160.327
C04263=1015.386,73.773,-115.987,166.273,56.795,160.328
C04264=1015.381,73.524,-115.971,166.269,56.805,160.329
C04265=1015.376,73.274,-115.955,166.268,56.815,160.331
C04266=1015.371,73.024,-115.940,166.265,56.825,160.332
C04267=1015.366,72.775,-115.924,166.263,56.834,160.333
C04268=1015.362,72.526,-115.908,166.260,56.844,160.334
C04269=1015.357,72.277,-115.892,166.257,56.854,160.336
C04270=1015.352,72.027,-115.877,166.255,56.863,160.337
C04271=1015.347,71.777,-115.861,166.252,56.873,160.338
C04272=1015.342,71.528,-115.845,166.250,56.883,160.340
C04273=1015.338,71.278,-115.829,166.248,56.893,160.341
C04274=1015.333,71.029,-115.814,166.246,56.902,160.342
C04275=1015.328,70.779,-115.797,166.242,56.912,160.343
C04276=1015.323,70.530,-115.782,166.240,56.922,160.345
C04277=1015.318,70.281,-115.766,166.238,56.931,160.346
C04278=1015.313,70.031,-115.751,166.236,56.941,160.347
C04279=1015.309,69.782,-115.735,166.232,56.951,160.349
C04280=1015.303,69.532,-115.719,166.230,56.960,160.350
C04281=1015.299,69.283,-115.703,166.228,56.970,160.351
C04282=1015.294,69.033,-115.687,166.226,56.979,160.353
C04283=1015.289,68.784,-115.672,166.222,56.989,160.354
C04284=1015.285,68.535,-115.656,166.220,56.999,160.355
C04285=1015.280,68.285,-115.641,166.218,57.008,160.356
C04286=1015.275,68.035,-115.625,166.216,57.018,160.358
C04287=1015.270,67.786,-115.610,166.213,57.029,160.359
C04288=1015.266,67.536,-115.594,166.211,57.038,160.360
C04289=1015.260,67.287,-115.578,166.209,57.048,160.362
C04290=1015.255,67.038,-115.563,166.206,57.057,160.363
C04291=1015.251,66.789,-115.547,166.203,57.067,160.364
C04292=1015.245,66.539,-115.532,166.201,57.077,160.366
C04293=1015.241,66.289,-115.516,166.199,57.086,160.367
C04294=1015.236,66.040,-115.501,166.195,57.096,160.368
C04295=1015.231,65.791,-115.485,166.193,57.106,160.369
C04296=1015.227,65.541,-115.470,166.191,57.115,160.371
C04297=1015.222,65.292,-115.454,166.189,57.125,160.372
C04298=1015.217,65.042,-115.439,166.185,57.135,160.373
C04299=1015.212,64.792,-115.423,166.183,57.144,160.374
C04300=1015.207,64.543,-115.408,166.181,57.154,160.376
C04301=1015.202,64.293,-115.392,166.179,57.163,160.377
C04302=1015.197,64.044,-115.377,166.176,57.173,160.378
C04303=1015.192,63.795,-115.362,166.173,57.183,160.380
C04304=1015.188,63.545,-115.346,166.171,57.193,160.381
C04305=1015.183,63.295,-115.332,166.169,57.202,160.382
C04306=1015.178,63.046,-115.316,166.167,57.212,160.384
C04307=1015.174,62.796,-115.301,166.164,57.222,160.385
C04308=1015.168,62.546,-115.285,166.162,57.231,160.386
C04309=1015.163,62.297,-115.270,166.159,57.241,160.387
C04310=1015.158,62.048,-115.255,166.157,57.252,160.389
C04311=1015.153,61.798,-115.240,166.155,57.261,160.390
C04312=1015.148,61.549,-115.225,166.152,57.271,160.392
C04313=1015.143,61.300,-115.210,166.149,57.281,160.393
C04314=1015.138,61.050,-115.195,166.147,57.290,160.394
C04315=1015.134,60.800,-115.180,166.145,57.300,160.395
C04316=1015.128,60.551,-115.165,166.142,57.310,160.396
C04317=1015.123,60.302,-115.150,166.139,57.319,160.398
C04318=1015.118,60.053,-115.135,166.137,57.329,160.399
C04319=1015.114,59.803,-115.120,166.135,57.340,160.401
C04320=1015.108,59.553,-115.105,166.133,57.349,160.402
C04321=1015.103,59.303,-115.090,166.130,57.359,160.403
C04322=1015.099,59.053,-115.075,166.128,57.368,160.405
C04323=1015.093,58.773,-115.058,166.125,57.380,160.406
C04324=1015.088,58.493,-115.041,166.122,57.390,160.407
C04325=1015.082,58.211,-115.024,166.119,57.401,160.409
C04326=1015.077,57.931,-115.007,166.117,57.412,160.410
C04327=1015.072,57.681,-114.993,166.114,57.422,160.411
C04328=1015.067,57.432,-114.977,166.111,57.431,160.413
C04329=1015.062,57.183,-114.962,166.109,57.441,160.414
C04330=1015.057,56.933,-114.948,166.107,57.451,160.415
C04331=1015.052,56.683,-114.933,166.104,57.461,160.417
C04332=1015.047,56.434,-114.917,166.102,57.470,160.418
C04333=1015.042,56.184,-114.903,166.100,57.480,160.419
C04334=1015.037,55.935,-114.888,166.098,57.489,160.421
C04335=1015.032,55.685,-114.873,166.096,57.499,160.422
C04336=1015.027,55.436,-114.858,166.092,57.509,160.423
C04337=1015.022,55.187,-114.843,166.090,57.519,160.425
C04338=1015.018,54.937,-114.829,166.088,57.528,160.426
C04339=1015.013,54.687,-114.813,166.086,57.538,160.427
C04340=1015.007,54.438,-114.798,166.082,57.547,160.428
C04341=1015.003,54.188,-114.784,166.080,57.557,160.429
C04342=1014.998,53.939,-114.769,166.078,57.566,160.431
C04343=1014.993,53.689,-114.754,166.076,57.576,160.432
C04344=1014.988,53.440,-114.739,166.074,57.586,160.434
C04345=1014.983,53.190,-114.724,166.072,57.595,160.435
C04346=1014.978,52.941,-114.709,166.068,57.605,160.436
C04347=1014.973,52.691,-114.694,166.066,57.614,160.437
C04348=1014.968,52.442,-114.680,166.064,57.624,160.438
C04349=1014.963,52.192,-114.664,166.062,57.633,160.440
C04350=1014.959,51.943,-114.650,166.060,57.643,160.441
C04351=1014.954,51.694,-114.635,166.057,57.652,160.442
C04352=1014.949,51.444,-114.621,166.054,57.662,160.443
C04353=1014.944,51.195,-114.606,166.052,57.672,160.445
C04354=1014.940,50.945,-114.591,166.050,57.681,160.446
C04355=1014.935,50.695,-114.576,166.047,57.690,160.447
C04356=1014.930,50.446,-114.561,166.045,57.700,160.449
C04357=1014.925,50.196,-114.546,166.043,57.709,160.450
C04358=1014.920,49.946,-114.532,166.041,57.718,160.451
C04359=1014.915,49.697,-114.517,166.039,57.728,160.452
C04360=1014.911,49.447,-114.502,166.037,57.738,160.454
C04361=1014.907,49.198,-114.487,166.033,57.747,160.455
C04362=1014.902,48.949,-114.472,166.031,57.757,160.456
C04363=1014.897,48.699,-114.457,166.029,57.766,160.457
C04364=1014.892,48.449,-114.443,166.026,57.775,160.458
C04365=1014.887,48.200,-114.428,166.024,57.785,160.460
C04366=1014.882,47.950,-114.413,166.022,57.794,160.461
C04367=1014.877,47.701,-114.398,166.019,57.803,160.462
C04368=1014.872,47.451,-114.383,166.017,57.813,160.464
C04369=1014.868,47.202,-114.369,166.015,57.822,160.465
C04370=1014.863,46.953,-114.354,166.013,57.831,160.466
C04371=1014.859,46.703,-114.340,166.010,57.840,160.467
C04372=1014.854,46.453,-114.325,166.008,57.850,160.468
C04373=1014.849,46.204,-114.310,166.005,57.859,160.469
C04374=1014.844,45.954,-114.295,166.003,57.869,160.471
C04375=1014.839,45.704,-114.280,166.001,57.878,160.472
C04376=1014.835,45.455,-114.266,165.999,57.887,160.473
C04377=1014.830,45.206,-114.251,165.997,57.897,160.475
C04378=1014.825,44.956,-114.237,165.994,57.906,160.476
C04379=1014.820,44.707,-114.222,165.992,57.915,160.477
C04380=1014.815,44.457,-114.207,165.990,57.924,160.478
C04381=1014.811,44.208,-114.193,165.987,57.933,160.479
C04382=1014.806,43.958,-114.178,165.985,57.943,160.481
C04383=1014.801,43.709,-114.163,165.982,57.952,160.482
C04384=1014.797,43.459,-114.149,165.980,57.962,160.483
C04385=1014.792,43.209,-114.134,165.978,57.971,160.484
C04386=1014.787,42.960,-114.120,165.976,57.980,160.486
C04387=1014.781,42.679,-114.103,165.973,57.990,160.487
C04388=1014.776,42.398,-114.086,165.970,58.000,160.488
C04389=1014.771,42.118,-114.070,165.968,58.011,160.490
C04390=1014.766,41.837,-114.053,165.965,58.021,160.491
C04391=1014.760,41.587,-114.040,165.963,58.031,160.492
C04392=1014.756,41.338,-114.026,165.961,58.040,160.493
C04393=1014.751,41.088,-114.011,165.958,58.050,160.494
C04394=1014.746,40.839,-113.996,165.956,58.059,160.496
C04395=1014.741,40.589,-113.982,165.953,58.068,160.497
C04396=1014.737,40.340,-113.968,165.951,58.078,160.498
C04397=1014.732,40.090,-113.953,165.949,58.087,160.499
C04398=1014.726,39.841,-113.940,165.946,58.096,160.500
C04399=1014.722,39.591,-113.925,165.944,58.106,160.502
C04400=1014.718,39.342,-113.911,165.942,58.115,160.503
C04401=1014.713,39.092,-113.896,165.940,58.124,160.504
C04402=1014.707,38.843,-113.882,165.937,58.133,160.505
C04403=1014.702,38.593,-113.868,165.935,58.143,160.507
C04404=1014.698,38.344,-113.853,165.933,58.152,160.508
C04405=1014.693,38.094,-113.840,165.930,58.161,160.509
C04406=1014.688,37.844,-113.825,165.928,58.170,160.510
C04407=1014.683,37.594,-113.811,165.925,58.179,160.511
C04408=1014.678,37.345,-113.797,165.924,58.189,160.513
C04409=1014.674,37.095,-113.783,165.921,58.198,160.514
C04410=1014.669,36.846,-113.768,165.918,58.207,160.515
C04411=1014.665,36.596,-113.754,165.917,58.217,160.516
C04412=1014.659,36.347,-113.740,165.915,58.225,160.518
C04413=1014.655,36.097,-113.726,165.912,58.234,160.519
C04414=1014.649,35.847,-113.712,165.910,58.244,160.520
C04415=1014.645,35.598,-113.698,165.907,58.253,160.521
C04416=1014.639,35.349,-113.684,165.905,58.263,160.522
C04417=1014.635,35.099,-113.670,165.903,58.272,160.524
C04418=1014.630,34.850,-113.656,165.901,58.282,160.525
C04419=1014.625,34.600,-113.642,165.898,58.291,160.526
C04420=1014.620,34.350,-113.628,165.896,58.300,160.527
C04421=1014.616,34.101,-113.614,165.894,58.309,160.528
C04422=1014.610,33.851,-113.601,165.891,58.318,160.530
C04423=1014.606,33.601,-113.586,165.889,58.328,160.531
C04424=1014.601,33.352,-113.573,165.887,58.337,160.532
C04425=1014.595,33.103,-113.559,165.884,58.346,160.533
C04426=1014.591,32.853,-113.544,165.882,58.356,160.535
C04427=1014.586,32.604,-113.531,165.880,58.365,160.536
C04428=1014.581,32.353,-113.517,165.877,58.374,160.537
C04429=1014.576,32.104,-113.503,165.875,58.384,160.538
C04430=1014.572,31.855,-113.489,165.873,58.393,160.539
C04431=1014.566,31.605,-113.475,165.871,58.401,160.541
C04432=1014.562,31.356,-113.461,165.869,58.410,160.542
C04433=1014.557,31.106,-113.447,165.867,58.420,160.543
C04434=1014.551,30.856,-113.434,165.865,58.429,160.544
C04435=1014.547,30.607,-113.420,165.862,58.438,160.545
C04436=1014.542,30.357,-113.406,165.860,58.447,160.546
C04437=1014.537,30.107,-113.392,165.857,58.456,160.547
C04438=1014.532,29.859,-113.378,165.855,58.466,160.549
C04439=1014.528,29.608,-113.364,165.853,58.475,160.550
C04440=1014.523,29.359,-113.351,165.850,58.484,160.551
C04441=1014.518,29.109,-113.336,165.848,58.493,160.552
C04442=1014.513,28.860,-113.323,165.845,58.502,160.553
C04443=1014.509,28.610,-113.309,165.844,58.510,160.555
C04444=1014.503,28.360,-113.295,165.842,58.520,160.556
C04445=1014.498,28.112,-113.282,165.840,58.529,160.557
C04446=1014.494,27.862,-113.267,165.837,58.538,160.558
C04447=1014.489,27.612,-113.255,165.835,58.547,160.559
C04448=1014.484,27.362,-113.240,165.832,58.556,160.560
C04449=1014.479,27.113,-113.226,165.830,58.565,160.561
C04450=1014.474,26.863,-113.214,165.827,58.574,160.563
C04451=1014.469,26.582,-113.198,165.826,58.584,160.564
C04452=1014.464,26.302,-113.182,165.823,58.595,160.566
C04453=1014.458,26.021,-113.167,165.820,58.605,160.567
C04454=1014.452,25.741,-113.151,165.817,58.615,160.568
C04455=1014.448,25.491,-113.139,165.816,58.624,160.569
C04456=1014.442,25.242,-113.125,165.814,58.633,160.570
C04457=1014.438,24.992,-113.111,165.811,58.642,160.571
C04458=1014.433,24.742,-113.097,165.809,58.651,160.573
C04459=1014.428,24.493,-113.085,165.807,58.660,160.574
C04460=1014.423,24.243,-113.071,165.804,58.670,160.575
C04461=1014.418,23.994,-113.058,165.802,58.679,160.576
C04462=1014.413,23.744,-113.044,165.799,58.688,160.577
C04463=1014.409,23.495,-113.030,165.797,58.697,160.578
C04464=1014.403,23.245,-113.017,165.796,58.705,160.580
C04465=1014.399,22.996,-113.003,165.793,58.714,160.581
C04466=1014.393,22.746,-112.990,165.791,58.723,160.582
C04467=1014.389,22.497,-112.976,165.788,58.732,160.583
C04468=1014.384,22.246,-112.963,165.786,58.741,160.584
C04469=1014.379,21.997,-112.950,165.784,58.750,160.585
C04470=1014.374,21.747,-112.936,165.782,58.759,160.587
C04471=1014.369,21.498,-112.924,165.780,58.768,160.588
C04472=1014.365,21.248,-112.909,165.777,58.777,160.589
C04473=1014.360,20.998,-112.896,165.775,58.786,160.590
C04474=1014.355,20.749,-112.882,165.773,58.795,160.591
C04475=1014.350,20.499,-112.870,165.771,58.804,160.592
C04476=1014.345,20.250,-112.856,165.769,58.813,160.593
C04477=1014.341,20.000,-112.842,165.766,58.821,160.594
C04478=1014.336,19.751,-112.829,165.763,58.830,160.595
C04479=1014.331,19.501,-112.816,165.761,58.839,160.597
C04480=1014.326,19.251,-112.803,165.760,58.848,160.598
C04481=1014.321,19.002,-112.789,165.757,58.857,160.599
C04482=1014.317,18.752,-112.776,165.755,58.866,160.600
C04483=1014.311,18.502,-112.762,165.752,58.875,160.601
C04484=1014.307,18.253,-112.749,165.751,58.884,160.603
C04485=1014.302,18.003,-112.736,165.748,58.892,160.603
C04486=1014.297,17.754,-112.722,165.746,58.901,160.604
C04487=1014.292,17.504,-112.710,165.743,58.910,160.606
C04488=1014.287,17.254,-112.697,165.741,58.919,160.607
C04489=1014.282,17.005,-112.684,165.740,58.928,160.608
C04490=1014.277,16.755,-112.670,165.737,58.937,160.609
C04491=1014.272,16.506,-112.657,165.735,58.946,160.610
C04492=1014.268,16.256,-112.644,165.732,58.954,160.611
C04493=1014.262,16.007,-112.630,165.730,58.963,160.612
C04494=1014.258,15.757,-112.618,165.728,58.972,160.613
C04495=1014.253,15.507,-112.605,165.726,58.981,160.615
C04496=1014.248,15.257,-112.592,165.723,58.989,160.615
C04497=1014.243,15.008,-112.578,165.721,58.998,160.617
C04498=1014.238,14.758,-112.565,165.719,59.007,160.618
C04499=1014.233,14.509,-112.552,165.717,59.016,160.619
C04500=1014.229,14.259,-112.540,165.715,59.024,160.620
C04501=1014.223,14.010,-112.526,165.712,59.033,160.621
C04502=1014.219,13.760,-112.513,165.710,59.042,160.622
C04503=1014.214,13.510,-112.500,165.708,59.050,160.623
C04504=1014.210,13.260,-112.486,165.706,59.059,160.624
C04505=1014.205,13.011,-112.474,165.703,59.068,160.625
C04506=1014.199,12.761,-112.461,165.700,59.076,160.626
C04507=1014.195,12.511,-112.448,165.699,59.085,160.628
C04508=1014.190,12.262,-112.435,165.697,59.094,160.629
C04509=1014.185,12.012,-112.422,165.694,59.103,160.630
C04510=1014.179,11.763,-112.409,165.692,59.112,160.631
C04511=1014.175,11.514,-112.397,165.690,59.120,160.632
C04512=1014.170,11.263,-112.384,165.688,59.129,160.633
C04513=1014.165,11.014,-112.371,165.685,59.138,160.634
C04514=1014.160,10.765,-112.359,165.683,59.148,160.635
C04515=1014.154,10.484,-112.344,165.681,59.157,160.637
C04516=1014.149,10.206,-112.330,165.678,59.167,160.638
C04517=1014.143,9.927,-112.316,165.676,59.176,160.639
C04518=1014.138,9.648,-112.302,165.673,59.186,160.640
C04519=1014.133,9.399,-112.289,165.672,59.195,160.642
C04520=1014.128,9.148,-112.276,165.669,59.203,160.642
C04521=1014.124,8.898,-112.264,165.666,59.212,160.643
C04522=1014.118,8.649,-112.251,165.664,59.220,160.644
C04523=1014.114,8.400,-112.239,165.662,59.229,160.646
C04524=1014.108,8.149,-112.225,165.660,59.239,160.647
C04525=1014.104,7.900,-112.213,165.658,59.246,160.648
C04526=1014.099,7.651,-112.200,165.656,59.256,160.649
C04527=1014.094,7.401,-112.188,165.653,59.264,160.650
C04528=1014.089,7.151,-112.175,165.651,59.273,160.651
C04529=1014.084,6.902,-112.162,165.648,59.281,160.652
C04530=1014.079,6.652,-112.150,165.646,59.290,160.653
C04531=1014.074,6.403,-112.137,165.644,59.298,160.654
C04532=1014.069,6.153,-112.124,165.642,59.307,160.655
C04533=1014.064,5.904,-112.111,165.640,59.315,160.656
C04534=1014.060,5.653,-112.099,165.638,59.324,160.657
C04535=1014.055,5.404,-112.087,165.635,59.332,160.658
C04536=1014.050,5.154,-112.073,165.634,59.341,160.659
C04537=1014.045,4.905,-112.061,165.631,59.350,160.660
C04538=1014.040,4.655,-112.048,165.629,59.357,160.661
C04539=1014.035,4.406,-112.036,165.627,59.367,160.662
C04540=1014.031,4.156,-112.023,165.625,59.374,160.663
C04541=1014.025,3.906,-112.010,165.622,59.383,160.664
C04542=1014.021,3.656,-111.998,165.621,59.392,160.666
C04543=1014.016,3.407,-111.985,165.618,59.400,160.666
C04544=1014.012,3.157,-111.973,165.616,59.408,160.667
C04545=1014.006,2.908,-111.961,165.613,59.417,160.669
C04546=1014.002,2.658,-111.948,165.612,59.425,160.670
C04547=1013.997,2.408,-111.935,165.609,59.433,160.670
C04548=1013.992,2.158,-111.923,165.607,59.441,160.671
C04549=1013.987,1.909,-111.910,165.605,59.450,160.673
C04550=1013.982,1.659,-111.898,165.603,59.458,160.674
C04551=1013.978,1.410,-111.885,165.600,59.467,160.674
C04552=1013.973,1.161,-111.873,165.598,59.475,160.675
C04553=1013.968,0.910,-111.860,165.596,59.484,160.677
C04554=1013.963,0.660,-111.847,165.594,59.492,160.678
C04555=1013.959,0.411,-111.835,165.591,59.500,160.678
C04556=1013.953,0.162,-111.822,165.589,59.508,160.679
C04557=1013.949,-0.088,-111.810,165.587,59.516,160.681
C04558=1013.944,-0.338,-111.798,165.584,59.524,160.681
C04559=1013.940,-0.587,-111.785,165.582,59.532,160.682
C04560=1013.934,-0.837,-111.772,165.580,59.541,160.683
C04561=1013.929,-1.087,-111.759,165.578,59.549,160.685
C04562=1013.925,-1.337,-111.747,165.577,59.557,160.686
C04563=1013.920,-1.586,-111.735,165.574,59.566,160.686
C04564=1013.915,-1.835,-111.722,165.572,59.574,160.687
C04565=1013.911,-2.086,-111.710,165.570,59.582,160.688
C04566=1013.906,-2.335,-111.698,165.567,59.590,160.689
C04567=1013.901,-2.584,-111.685,165.565,59.598,160.690
C04568=1013.897,-2.834,-111.673,165.563,59.606,160.691
C04569=1013.892,-3.084,-111.660,165.561,59.614,160.692
C04570=1013.887,-3.333,-111.648,165.559,59.622,160.693
C04571=1013.882,-3.583,-111.635,165.556,59.630,160.694
C04572=1013.878,-3.833,-111.623,165.553,59.638,160.695
C04573=1013.873,-4.083,-111.610,165.551,59.646,160.696
C04574=1013.868,-4.332,-111.598,165.550,59.654,160.697
C04575=1013.863,-4.582,-111.586,165.548,59.662,160.698
C04576=1013.859,-4.832,-111.573,165.545,59.670,160.699
C04577=1013.854,-5.081,-111.562,165.543,59.678,160.700
C04578=1013.849,-5.331,-111.550,165.540,59.687,160.700
C04579=1013.844,-5.608,-111.536,165.538,59.696,160.702
C04580=1013.838,-5.885,-111.523,165.536,59.705,160.703
C04581=1013.832,-6.162,-111.510,165.534,59.714,160.704
C04582=1013.827,-6.439,-111.496,165.531,59.723,160.705
C04583=1013.822,-6.688,-111.484,165.529,59.732,160.706
C04584=1013.817,-6.938,-111.473,165.527,59.740,160.707
C04585=1013.813,-7.187,-111.460,165.524,59.747,160.708
C04586=1013.808,-7.437,-111.449,165.521,59.755,160.708
C04587=1013.803,-7.687,-111.437,165.520,59.763,160.710
C04588=1013.798,-7.937,-111.424,165.518,59.771,160.711
C04589=1013.793,-8.186,-111.413,165.515,59.780,160.711
C04590=1013.788,-8.436,-111.401,165.513,59.788,160.712
C04591=1013.783,-8.686,-111.389,165.511,59.796,160.713
C04592=1013.778,-8.935,-111.377,165.509,59.804,160.714
C04593=1013.773,-9.185,-111.365,165.507,59.812,160.715
C04594=1013.769,-9.435,-111.353,165.505,59.820,160.716
C04595=1013.764,-9.685,-111.341,165.503,59.827,160.717
C04596=1013.759,-9.934,-111.329,165.500,59.836,160.718
C04597=1013.754,-10.184,-111.317,165.498,59.844,160.719
C04598=1013.749,-10.434,-111.306,165.496,59.852,160.720
C04599=1013.745,-10.683,-111.293,165.494,59.860,160.721
C04600=1013.740,-10.933,-111.281,165.491,59.867,160.721
C04601=1013.735,-11.183,-111.270,165.489,59.875,160.723
C04602=1013.730,-11.432,-111.257,165.487,59.883,160.724
C04603=1013.725,-11.682,-111.246,165.485,59.891,160.724
C04604=1013.721,-11.931,-111.235,165.482,59.899,160.725
C04605=1013.716,-12.181,-111.223,165.480,59.907,160.726
C04606=1013.711,-12.430,-111.210,165.478,59.914,160.727
C04607=1013.706,-12.680,-111.199,165.476,59.922,160.728
C04608=1013.702,-12.930,-111.187,165.474,59.930,160.729
C04609=1013.697,-13.179,-111.175,165.472,59.938,160.730
C04610=1013.692,-13.429,-111.163,165.469,59.946,160.730
C04611=1013.687,-13.679,-111.151,165.467,59.954,160.732
C04612=1013.682,-13.929,-111.140,165.465,59.961,160.732
C04613=1013.677,-14.178,-111.127,165.463,59.969,160.733
C04614=1013.673,-14.429,-111.115,165.461,59.976,160.734
C04615=1013.668,-14.678,-111.104,165.459,59.984,160.735
C04616=1013.663,-14.927,-111.093,165.456,59.992,160.736
C04617=1013.659,-15.177,-111.080,165.455,60.000,160.737
C04618=1013.654,-15.427,-111.068,165.451,60.007,160.737
C04619=1013.649,-15.677,-111.057,165.449,60.015,160.738
C04620=1013.645,-15.927,-111.045,165.447,60.023,160.739
C04621=1013.640,-16.176,-111.033,165.445,60.031,160.740
C04622=1013.635,-16.426,-111.022,165.443,60.038,160.741
C04623=1013.630,-16.676,-111.011,165.441,60.046,160.742
C04624=1013.625,-16.925,-110.999,165.439,60.053,160.743
C04625=1013.620,-17.175,-110.988,165.437,60.061,160.744
C04626=1013.615,-17.425,-110.976,165.434,60.069,160.744
C04627=1013.611,-17.675,-110.964,165.432,60.077,160.745
C04628=1013.606,-17.925,-110.953,165.429,60.084,160.746
C04629=1013.601,-18.174,-110.941,165.428,60.092,160.747
C04630=1013.596,-18.424,-110.930,165.425,60.099,160.748
C04631=1013.591,-18.673,-110.919,165.424,60.107,160.749
C04632=1013.586,-18.923,-110.907,165.421,60.115,160.749
C04633=1013.581,-19.173,-110.896,165.419,60.123,160.750
C04634=1013.576,-19.423,-110.884,165.417,60.130,160.751
C04635=1013.572,-19.672,-110.873,165.415,60.137,160.752
C04636=1013.567,-19.922,-110.862,165.413,60.145,160.753
C04637=1013.562,-20.171,-110.850,165.410,60.153,160.754
C04638=1013.557,-20.421,-110.839,165.409,60.161,160.755
C04639=1013.552,-20.671,-110.827,165.405,60.168,160.755
C04640=1013.548,-20.920,-110.816,165.403,60.176,160.756
C04641=1013.543,-21.170,-110.805,165.401,60.184,160.757
C04642=1013.538,-21.420,-110.793,165.399,60.191,160.758
C04643=1013.533,-21.695,-110.781,165.397,60.199,160.759
C04644=1013.527,-21.970,-110.768,165.394,60.207,160.760
C04645=1013.522,-22.245,-110.755,165.393,60.215,160.761
C04646=1013.517,-22.520,-110.743,165.389,60.223,160.761
C04647=1013.512,-22.770,-110.732,165.387,60.231,160.762
C04648=1013.507,-23.020,-110.721,165.385,60.238,160.763
C04649=1013.503,-23.269,-110.710,165.383,60.246,160.764
C04650=1013.498,-23.519,-110.698,165.380,60.253,160.764
C04651=1013.493,-23.769,-110.687,165.379,60.260,160.765
C04652=1013.488,-24.018,-110.676,165.377,60.267,160.766
C04653=1013.483,-24.268,-110.664,165.374,60.274,160.767
C04654=1013.478,-24.518,-110.653,165.372,60.282,160.768
C04655=1013.473,-24.767,-110.641,165.370,60.290,160.768
C04656=1013.469,-25.017,-110.631,165.368,60.297,160.769
C04657=1013.465,-25.267,-110.619,165.365,60.304,160.770
C04658=1013.460,-25.517,-110.607,165.363,60.312,160.771
C04659=1013.456,-25.766,-110.596,165.362,60.318,160.771
C04660=1013.451,-26.016,-110.585,165.359,60.326,160.772
C04661=1013.446,-26.266,-110.573,165.357,60.333,160.773
C04662=1013.442,-26.515,-110.563,165.355,60.340,160.774
C04663=1013.437,-26.765,-110.551,165.352,60.348,160.774
C04664=1013.432,-27.015,-110.540,165.351,60.354,160.775
C04665=1013.427,-27.264,-110.529,165.349,60.362,160.776
C04666=1013.422,-27.514,-110.517,165.345,60.368,160.776
C04667=1013.417,-27.764,-110.507,165.343,60.375,160.777
C04668=1013.412,-28.014,-110.495,165.341,60.383,160.778
C04669=1013.408,-28.263,-110.484,165.339,60.390,160.779
C04670=1013.403,-28.514,-110.473,165.337,60.397,160.779
C04671=1013.398,-28.763,-110.463,165.335,60.404,160.780
C04672=1013.394,-29.013,-110.452,165.332,60.411,160.781
C04673=1013.389,-29.263,-110.441,165.330,60.419,160.782
C04674=1013.384,-29.512,-110.429,165.328,60.426,160.782
C04675=1013.379,-29.762,-110.419,165.326,60.433,160.783
C04676=1013.374,-30.012,-110.408,165.324,60.440,160.784
C04677=1013.370,-30.261,-110.397,165.322,60.448,160.785
C04678=1013.365,-30.511,-110.386,165.319,60.455,160.785
C04679=1013.359,-30.760,-110.375,165.317,60.462,160.786
C04680=1013.355,-31.010,-110.365,165.316,60.469,160.787
C04681=1013.350,-31.260,-110.353,165.313,60.476,160.787
C04682=1013.346,-31.510,-110.343,165.310,60.483,160.788
C04683=1013.340,-31.759,-110.332,165.309,60.490,160.789
C04684=1013.336,-32.009,-110.322,165.307,60.497,160.790
C04685=1013.331,-32.259,-110.310,165.304,60.504,160.790
C04686=1013.327,-32.509,-110.300,165.301,60.511,160.791
C04687=1013.321,-32.758,-110.289,165.300,60.518,160.792
C04688=1013.316,-33.009,-110.278,165.298,60.525,160.792
C04689=1013.312,-33.258,-110.267,165.295,60.532,160.793
C04690=1013.307,-33.508,-110.256,165.293,60.538,160.794
C04691=1013.302,-33.757,-110.246,165.291,60.546,160.795
C04692=1013.297,-34.007,-110.235,165.288,60.552,160.795
C04693=1013.293,-34.256,-110.224,165.287,60.559,160.796
C04694=1013.288,-34.507,-110.213,165.284,60.566,160.797
C04695=1013.283,-34.756,-110.203,165.283,60.572,160.797
C04696=1013.278,-35.006,-110.192,165.280,60.580,160.798
C04697=1013.274,-35.255,-110.181,165.277,60.586,160.798
C04698=1013.269,-35.506,-110.170,165.276,60.593,160.799
C04699=1013.265,-35.755,-110.160,165.274,60.601,160.800
C04700=1013.260,-36.005,-110.149,165.272,60.607,160.800
C04701=1013.255,-36.255,-110.138,165.269,60.614,160.801
C04702=1013.250,-36.504,-110.127,165.267,60.620,160.802
C04703=1013.246,-36.754,-110.117,165.265,60.627,160.802
C04704=1013.241,-37.004,-110.106,165.263,60.633,160.803
C04705=1013.236,-37.253,-110.095,165.260,60.640,160.803
C04706=1013.232,-37.504,-110.084,165.259,60.647,160.804
C04707=1013.226,-37.777,-110.073,165.257,60.654,160.805
C04708=1013.221,-38.052,-110.061,165.254,60.662,160.806
C04709=1013.216,-38.326,-110.049,165.252,60.669,160.807
C04710=1013.211,-38.600,-110.037,165.249,60.675,160.807
C04711=1013.206,-38.849,-110.027,165.247,60.683,160.808
C04712=1013.202,-39.099,-110.016,165.245,60.689,160.808
C04713=1013.197,-39.348,-110.005,165.242,60.695,160.809
C04714=1013.192,-39.598,-109.995,165.240,60.702,160.810
C04715=1013.187,-39.848,-109.984,165.237,60.709,160.810
C04716=1013.183,-40.098,-109.975,165.235,60.715,160.810
C04717=1013.178,-40.348,-109.963,165.233,60.722,160.811
C04718=1013.173,-40.597,-109.953,165.231,60.728,160.812
C04719=1013.168,-40.847,-109.943,165.229,60.736,160.813
C04720=1013.163,-41.097,-109.933,165.227,60.742,160.813
C04721=1013.159,-41.346,-109.922,165.225,60.748,160.814
C04722=1013.154,-41.597,-109.912,165.223,60.755,160.814
///RCONF 1,0,0,1,0,0,0,0,0,0,0,0,0,0,0,0,0,0,0,0,0,0,0,0
C04723=1013.150,-41.846,-109.902,165.221,60.761,160.815
C04724=1013.145,-42.095,-109.891,165.218,60.768,160.815
C04725=1013.140,-42.346,-109.881,165.216,60.774,160.816
C04726=1013.135,-42.595,-109.871,165.214,60.781,160.817
C04727=1013.130,-42.845,-109.860,165.212,60.788,160.817
C04728=1013.125,-43.095,-109.850,165.210,60.794,160.818
C04729=1013.121,-43.344,-109.840,165.207,60.800,160.818
C04730=1013.116,-43.595,-109.830,165.205,60.806,160.819
C04731=1013.112,-43.844,-109.819,165.203,60.813,160.819
C04732=1013.107,-44.093,-109.809,165.201,60.820,160.820
C04733=1013.101,-44.343,-109.799,165.199,60.826,160.821
C04734=1013.097,-44.593,-109.788,165.197,60.832,160.821
C04735=1013.092,-44.842,-109.778,165.194,60.839,160.822
C04736=1013.088,-45.093,-109.768,165.192,60.845,160.822
C04737=1013.083,-45.342,-109.758,165.190,60.851,160.823
C04738=1013.079,-45.592,-109.748,165.187,60.858,160.823
C04739=1013.073,-45.842,-109.737,165.185,60.864,160.824
C04740=1013.069,-46.092,-109.727,165.183,60.870,160.824
C04741=1013.064,-46.341,-109.717,165.181,60.876,160.825
C04742=1013.060,-46.592,-109.706,165.179,60.882,160.826
C04743=1013.055,-46.841,-109.697,165.176,60.889,160.826
C04744=1013.051,-47.091,-109.686,165.174,60.895,160.827
C04745=1013.045,-47.341,-109.676,165.172,60.901,160.827
C04746=1013.041,-47.590,-109.666,165.171,60.907,160.828
C04747=1013.036,-47.840,-109.656,165.168,60.912,160.828
C04748=1013.031,-48.090,-109.646,165.165,60.919,160.828
C04749=1013.027,-48.340,-109.635,165.163,60.925,160.829
C04750=1013.022,-48.589,-109.626,165.161,60.931,160.830
C04751=1013.018,-48.839,-109.615,165.159,60.937,160.830
C04752=1013.013,-49.089,-109.605,165.157,60.943,160.831
C04753=1013.008,-49.339,-109.595,165.155,60.949,160.831
C04754=1013.004,-49.588,-109.585,165.153,60.955,160.832
C04755=1012.999,-49.838,-109.574,165.151,60.961,160.832
C04756=1012.994,-50.088,-109.564,165.149,60.967,160.833
C04757=1012.990,-50.338,-109.554,165.145,60.973,160.833
C04758=1012.985,-50.587,-109.544,165.143,60.979,160.833
C04759=1012.981,-50.837,-109.534,165.141,60.985,160.834
C04760=1012.976,-51.087,-109.523,165.139,60.991,160.834
C04761=1012.971,-51.336,-109.514,165.137,60.997,160.835
C04762=1012.967,-51.587,-109.504,165.135,61.003,160.835
C04763=1012.962,-51.837,-109.494,165.133,61.009,160.836
C04764=1012.957,-52.086,-109.484,165.131,61.015,160.836
C04765=1012.952,-52.336,-109.475,165.129,61.021,160.837
C04766=1012.947,-52.586,-109.465,165.127,61.027,160.837
C04767=1012.943,-52.835,-109.455,165.125,61.033,160.838
C04768=1012.938,-53.085,-109.446,165.121,61.039,160.838
C04769=1012.933,-53.335,-109.436,165.119,61.045,160.839
C04770=1012.928,-53.584,-109.426,165.117,61.051,160.839
C04771=1012.921,-53.919,-109.414,165.114,61.059,160.840
C04772=1012.915,-54.254,-109.401,165.112,61.066,160.840
C04773=1012.908,-54.588,-109.388,165.108,61.074,160.841
C04774=1012.902,-54.922,-109.375,165.106,61.083,160.842
C04775=1012.898,-55.172,-109.365,165.103,61.088,160.842
C04776=1012.893,-55.422,-109.356,165.101,61.094,160.842
C04777=1012.888,-55.672,-109.346,165.099,61.100,160.843
C04778=1012.883,-55.922,-109.337,165.097,61.106,160.843
C04779=1012.878,-56.171,-109.327,165.094,61.111,160.844
C04780=1012.874,-56.421,-109.318,165.092,61.117,160.844
C04781=1012.869,-56.671,-109.308,165.091,61.122,160.845
C04782=1012.864,-56.920,-109.299,165.089,61.128,160.845
C04783=1012.860,-57.170,-109.290,165.086,61.134,160.845
C04784=1012.855,-57.419,-109.280,165.084,61.139,160.846
C04785=1012.850,-57.669,-109.271,165.082,61.145,160.846
C04786=1012.845,-57.920,-109.261,165.079,61.151,160.846
C04787=1012.845,-46.064,-110.150,165.165,61.118,160.868
C04788=1012.850,-45.813,-110.161,165.167,61.112,160.868
C04789=1012.855,-45.564,-110.170,165.169,61.106,160.867
C04790=1012.859,-45.314,-110.181,165.172,61.101,160.867
C04791=1012.864,-45.065,-110.191,165.174,61.095,160.866
C04792=1012.868,-44.814,-110.201,165.175,61.089,160.866
C04793=1012.873,-44.565,-110.211,165.178,61.083,160.865
C04794=1012.877,-44.315,-110.222,165.180,61.077,160.865
C04795=1012.883,-44.065,-110.232,165.182,61.071,160.864
C04796=1012.888,-43.816,-110.242,165.184,61.065,160.863
C04797=1012.892,-43.566,-110.252,165.186,61.059,160.863
C04798=1012.897,-43.316,-110.262,165.188,61.053,160.863
C04799=1012.901,-43.066,-110.272,165.191,61.047,160.862
C04800=1012.906,-42.817,-110.283,165.193,61.040,160.862
C04801=1012.911,-42.567,-110.294,165.195,61.034,160.861
C04802=1012.916,-42.317,-110.304,165.197,61.028,160.860
C04803=1012.920,-42.068,-110.314,165.199,61.022,160.860
C04804=1012.925,-41.818,-110.324,165.201,61.017,160.860
C04805=1012.930,-41.568,-110.335,165.203,61.011,160.859
///RCONF 1,0,0,0,0,0,0,0,0,0,0,0,0,0,0,0,0,0,0,0,0,0,0,0
C04806=1012.934,-41.318,-110.344,165.206,61.004,160.859
C04807=1012.939,-41.068,-110.355,165.208,60.998,160.858
C04808=1012.944,-40.819,-110.365,165.210,60.992,160.857
C04809=1012.949,-40.568,-110.376,165.212,60.986,160.857
C04810=1012.954,-40.319,-110.386,165.215,60.979,160.856
C04811=1012.958,-40.070,-110.397,165.217,60.973,160.856
C04812=1012.963,-39.820,-110.407,165.218,60.966,160.855
C04813=1012.967,-39.570,-110.417,165.220,60.960,160.854
C04814=1012.973,-39.320,-110.427,165.222,60.954,160.854
C04815=1012.977,-39.071,-110.438,165.225,60.948,160.854
C04816=1012.984,-38.686,-110.454,165.228,60.938,160.853
C04817=1012.991,-38.301,-110.471,165.231,60.928,160.852
C04818=1012.999,-37.918,-110.487,165.234,60.918,160.851
C04819=1013.006,-37.534,-110.504,165.238,60.909,160.850
C04820=1013.010,-37.284,-110.514,165.239,60.902,160.849
C04821=1013.015,-37.034,-110.525,165.241,60.896,160.849
C04822=1013.020,-36.785,-110.535,165.244,60.890,160.848
C04823=1013.024,-36.534,-110.546,165.246,60.884,160.848
C04824=1013.029,-36.285,-110.557,165.248,60.878,160.847
C04825=1013.033,-36.035,-110.568,165.251,60.871,160.847
C04826=1013.038,-35.785,-110.578,165.252,60.864,160.846
C04827=1013.043,-35.535,-110.589,165.254,60.858,160.845
C04828=1013.047,-35.286,-110.599,165.257,60.851,160.845
C04829=1013.052,-35.036,-110.611,165.259,60.845,160.844
C04830=1013.057,-34.787,-110.621,165.260,60.838,160.843
C04831=1013.062,-34.537,-110.632,165.263,60.832,160.843
C04832=1013.066,-34.287,-110.643,165.265,60.826,160.842
C04833=1013.071,-34.037,-110.653,165.268,60.819,160.842
C04834=1013.076,-33.788,-110.664,165.269,60.812,160.841
C04835=1013.081,-33.537,-110.675,165.271,60.806,160.840
C04836=1013.085,-33.288,-110.686,165.273,60.799,160.839
C04837=1013.090,-33.038,-110.697,165.275,60.793,160.839
C04838=1013.095,-32.789,-110.707,165.278,60.786,160.838
C04839=1013.100,-32.539,-110.718,165.279,60.779,160.837
C04840=1013.104,-32.290,-110.729,165.282,60.773,160.837
C04841=1013.109,-32.039,-110.740,165.284,60.766,160.836
C04842=1013.114,-31.790,-110.750,165.287,60.759,160.836
C04843=1013.119,-31.540,-110.761,165.288,60.752,160.835
C04844=1013.123,-31.290,-110.771,165.291,60.746,160.834
C04845=1013.128,-31.040,-110.783,165.292,60.739,160.833
C04846=1013.132,-30.791,-110.793,165.295,60.732,160.833
C04847=1013.138,-30.541,-110.804,165.297,60.725,160.832
C04848=1013.143,-30.291,-110.816,165.299,60.719,160.832
C04849=1013.147,-30.042,-110.826,165.302,60.712,160.831
C04850=1013.152,-29.792,-110.837,165.303,60.705,160.830
C04851=1013.157,-29.543,-110.847,165.306,60.698,160.830
C04852=1013.162,-29.293,-110.859,165.308,60.691,160.829
C04853=1013.166,-29.043,-110.869,165.309,60.684,160.828
C04854=1013.171,-28.793,-110.880,165.312,60.677,160.828
C04855=1013.176,-28.543,-110.891,165.314,60.670,160.827
C04856=1013.180,-28.294,-110.902,165.316,60.663,160.826
C04857=1013.185,-28.044,-110.913,165.318,60.656,160.825
C04858=1013.190,-27.794,-110.924,165.320,60.650,160.825
C04859=1013.195,-27.545,-110.935,165.322,60.642,160.824
C04860=1013.199,-27.294,-110.946,165.325,60.636,160.823
C04861=1013.204,-27.045,-110.957,165.327,60.629,160.822
C04862=1013.209,-26.795,-110.968,165.329,60.622,160.822
C04863=1013.214,-26.546,-110.980,165.331,60.616,160.821
C04864=1013.218,-26.296,-110.990,165.333,60.608,160.820
C04865=1013.223,-26.046,-111.002,165.336,60.601,160.820
C04866=1013.228,-25.796,-111.013,165.337,60.594,160.819
C04867=1013.232,-25.547,-111.024,165.340,60.588,160.818
C04868=1013.237,-25.297,-111.036,165.342,60.580,160.818
C04869=1013.242,-25.047,-111.047,165.343,60.573,160.817
C04870=1013.246,-24.798,-111.058,165.346,60.566,160.816
C04871=1013.251,-24.548,-111.069,165.348,60.559,160.815
C04872=1013.256,-24.298,-111.081,165.350,60.553,160.815
C04873=1013.260,-24.049,-111.092,165.352,60.545,160.814
C04874=1013.265,-23.798,-111.103,165.355,60.538,160.813
C04875=1013.270,-23.549,-111.115,165.357,60.531,160.812
C04876=1013.274,-23.299,-111.126,165.358,60.524,160.811
C04877=1013.279,-23.050,-111.137,165.361,60.517,160.811
C04878=1013.284,-22.800,-111.149,165.363,60.509,160.810
C04879=1013.288,-22.551,-111.160,165.365,60.502,160.809
C04880=1013.294,-22.275,-111.172,165.368,60.495,160.809
C04881=1013.299,-22.001,-111.185,165.369,60.487,160.807
C04882=1013.304,-21.726,-111.197,165.373,60.479,160.807
C04883=1013.310,-21.451,-111.209,165.374,60.471,160.806
C04884=1013.315,-21.200,-111.220,165.377,60.464,160.805
C04885=1013.319,-20.951,-111.231,165.379,60.456,160.804
C04886=1013.324,-20.701,-111.243,165.381,60.449,160.804
C04887=1013.329,-20.452,-111.254,165.384,60.442,160.803
C04888=1013.333,-20.202,-111.266,165.385,60.435,160.802
C04889=1013.338,-19.952,-111.277,165.387,60.427,160.801
C04890=1013.343,-19.703,-111.289,165.389,60.419,160.800
C04891=1013.348,-19.453,-111.300,165.391,60.412,160.800
C04892=1013.353,-19.203,-111.312,165.394,60.405,160.799
C04893=1013.357,-18.954,-111.323,165.396,60.398,160.798
C04894=1013.362,-18.704,-111.334,165.398,60.390,160.797
C04895=1013.367,-18.454,-111.345,165.400,60.382,160.796
C04896=1013.372,-18.204,-111.357,165.402,60.375,160.796
C04897=1013.376,-17.955,-111.368,165.405,60.368,160.795
C04898=1013.381,-17.705,-111.379,165.407,60.360,160.794
C04899=1013.386,-17.455,-111.391,165.409,60.352,160.793
C04900=1013.391,-17.205,-111.402,165.411,60.345,160.792
C04901=1013.396,-16.956,-111.414,165.413,60.338,160.792
C04902=1013.401,-16.707,-111.425,165.415,60.330,160.791
C04903=1013.406,-16.457,-111.436,165.417,60.322,160.790
C04904=1013.410,-16.207,-111.448,165.420,60.315,160.789
C04905=1013.415,-15.957,-111.460,165.421,60.307,160.788
C04906=1013.420,-15.707,-111.471,165.423,60.300,160.787
C04907=1013.424,-15.457,-111.483,165.425,60.293,160.786
C04908=1013.429,-15.208,-111.495,165.427,60.286,160.786
C04909=1013.434,-14.959,-111.507,165.429,60.278,160.785
C04910=1013.438,-14.709,-111.519,165.432,60.270,160.784
C04911=1013.443,-14.459,-111.530,165.434,60.263,160.783
C04912=1013.448,-14.209,-111.542,165.436,60.255,160.782
C04913=1013.453,-13.959,-111.554,165.438,60.248,160.781
C04914=1013.458,-13.710,-111.566,165.440,60.241,160.781
C04915=1013.462,-13.461,-111.577,165.442,60.233,160.779
C04916=1013.466,-13.210,-111.589,165.444,60.225,160.779
C04917=1013.471,-12.961,-111.600,165.447,60.218,160.778
C04918=1013.477,-12.711,-111.613,165.448,60.210,160.777
C04919=1013.481,-12.461,-111.625,165.451,60.203,160.776
C04920=1013.486,-12.212,-111.636,165.453,60.195,160.775
C04921=1013.491,-11.962,-111.648,165.455,60.187,160.774
C04922=1013.495,-11.712,-111.660,165.458,60.179,160.774
C04923=1013.500,-11.463,-111.672,165.460,60.172,160.773
C04924=1013.505,-11.213,-111.683,165.462,60.164,160.772
C04925=1013.509,-10.963,-111.695,165.464,60.156,160.771
C04926=1013.514,-10.714,-111.707,165.466,60.148,160.770
C04927=1013.519,-10.464,-111.719,165.468,60.141,160.769
C04928=1013.524,-10.214,-111.731,165.470,60.133,160.768
C04929=1013.529,-9.964,-111.742,165.472,60.125,160.767
C04930=1013.534,-9.715,-111.755,165.475,60.117,160.767
C04931=1013.538,-9.465,-111.767,165.477,60.109,160.766
C04932=1013.543,-9.215,-111.778,165.479,60.102,160.765
C04933=1013.549,-8.966,-111.790,165.481,60.094,160.764
C04934=1013.552,-8.717,-111.802,165.483,60.086,160.763
C04935=1013.557,-8.467,-111.813,165.485,60.079,160.762
C04936=1013.562,-8.217,-111.825,165.488,60.070,160.761
C04937=1013.567,-7.968,-111.838,165.490,60.062,160.760
C04938=1013.572,-7.718,-111.849,165.491,60.054,160.759
C04939=1013.576,-7.468,-111.861,165.494,60.047,160.758
C04940=1013.581,-7.218,-111.873,165.497,60.039,160.758
C04941=1013.586,-6.969,-111.885,165.498,60.031,160.757
C04942=1013.591,-6.719,-111.897,165.500,60.023,160.755
C04943=1013.596,-6.469,-111.909,165.502,60.015,160.754
C04944=1013.601,-6.192,-111.922,165.505,60.006,160.754
C04945=1013.607,-5.916,-111.935,165.507,59.997,160.752
C04946=1013.612,-5.639,-111.949,165.510,59.989,160.752
C04947=1013.617,-5.363,-111.962,165.512,59.979,160.750
C04948=1013.622,-5.113,-111.973,165.515,59.971,160.750
C04949=1013.627,-4.863,-111.986,165.516,59.963,160.748
C04950=1013.632,-4.614,-111.998,165.518,59.955,160.747
C04951=1013.636,-4.363,-112.010,165.520,59.948,160.747
C04952=1013.641,-4.114,-112.023,165.523,59.939,160.746
C04953=1013.646,-3.865,-112.035,165.525,59.931,160.745
C04954=1013.651,-3.614,-112.047,165.527,59.923,160.744
C04955=1013.656,-3.364,-112.060,165.529,59.916,160.743
C04956=1013.660,-3.114,-112.072,165.531,59.908,160.742
C04957=1013.665,-2.865,-112.084,165.534,59.900,160.741
C04958=1013.670,-2.616,-112.097,165.536,59.892,160.740
C04959=1013.674,-2.366,-112.109,165.537,59.884,160.739
C04960=1013.679,-2.116,-112.121,165.540,59.876,160.738
C04961=1013.684,-1.867,-112.134,165.543,59.868,160.737
C04962=1013.688,-1.617,-112.146,165.544,59.860,160.736
C04963=1013.693,-1.367,-112.159,165.546,59.852,160.735
C04964=1013.698,-1.118,-112.171,165.548,59.844,160.734
C04965=1013.702,-0.868,-112.183,165.551,59.836,160.733
C04966=1013.707,-0.618,-112.196,165.552,59.828,160.732
C04967=1013.712,-0.369,-112.208,165.554,59.820,160.731
C04968=1013.717,-0.120,-112.221,165.557,59.811,160.731
C04969=1013.721,0.130,-112.233,165.559,59.803,160.729
C04970=1013.726,0.380,-112.246,165.561,59.795,160.728
C04971=1013.731,0.630,-112.258,165.564,59.787,160.728
C04972=1013.736,0.880,-112.270,165.565,59.779,160.727
C04973=1013.740,1.129,-112.283,165.567,59.771,160.725
C04974=1013.745,1.379,-112.296,165.570,59.762,160.725
C04975=1013.750,1.628,-112.308,165.572,59.754,160.724
C04976=1013.754,1.878,-112.320,165.573,59.746,160.723
C04977=1013.759,2.128,-112.333,165.576,59.738,160.722
C04978=1013.764,2.377,-112.345,165.578,59.730,160.721
C04979=1013.769,2.626,-112.358,165.581,59.722,160.720
C04980=1013.774,2.877,-112.370,165.583,59.714,160.719
C04981=1013.778,3.127,-112.383,165.584,59.705,160.717
C04982=1013.784,3.376,-112.395,165.587,59.697,160.717
C04983=1013.788,3.625,-112.408,165.589,59.689,160.716
C04984=1013.793,3.875,-112.421,165.591,59.680,160.715
C04985=1013.797,4.125,-112.433,165.593,59.672,160.714
C04986=1013.802,4.374,-112.445,165.595,59.663,160.713
C04987=1013.808,4.624,-112.458,165.597,59.655,160.711
C04988=1013.812,4.874,-112.471,165.600,59.647,160.711
C04989=1013.817,5.123,-112.484,165.602,59.639,160.710
C04990=1013.822,5.373,-112.495,165.604,59.630,160.708
C04991=1013.826,5.623,-112.508,165.606,59.622,160.707
C04992=1013.831,5.872,-112.521,165.609,59.613,160.707
C04993=1013.837,6.122,-112.533,165.610,59.605,160.705
C04994=1013.841,6.371,-112.546,165.613,59.596,160.704
C04995=1013.846,6.621,-112.559,165.615,59.588,160.703
C04996=1013.850,6.871,-112.571,165.617,59.579,160.702
C04997=1013.855,7.120,-112.583,165.619,59.571,160.701
C04998=1013.860,7.370,-112.596,165.622,59.563,160.700
C04999=1013.865,7.620,-112.609,165.624,59.554,160.699
C05000=1013.870,7.869,-112.622,165.626,59.546,160.698
C05001=1013.875,8.119,-112.634,165.628,59.536,160.697
C05002=1013.880,8.368,-112.647,165.630,59.528,160.696
C05003=1013.885,8.618,-112.660,165.632,59.519,160.695
C05004=1013.889,8.868,-112.672,165.635,59.511,160.694
C05005=1013.894,9.118,-112.684,165.636,59.502,160.693
C05006=1013.899,9.367,-112.697,165.639,59.494,160.692
C05007=1013.903,9.617,-112.710,165.640,59.485,160.690
C05008=1013.909,9.895,-112.724,165.644,59.476,160.689
C05009=1013.914,10.174,-112.739,165.646,59.466,160.688
C05010=1013.920,10.453,-112.753,165.648,59.456,160.687
C05011=1013.925,10.732,-112.767,165.651,59.447,160.686
C05012=1013.931,10.982,-112.779,165.653,59.438,160.685
C05013=1013.936,11.232,-112.792,165.655,59.429,160.684
C05014=1013.940,11.481,-112.805,165.657,59.421,160.682
C05015=1013.945,11.731,-112.818,165.659,59.412,160.681
C05016=1013.951,11.981,-112.830,165.662,59.403,160.680
C05017=1013.955,12.230,-112.843,165.663,59.395,160.679
C05018=1013.960,12.480,-112.856,165.666,59.386,160.678
C05019=1013.965,12.730,-112.869,165.668,59.376,160.677
C05020=1013.970,12.979,-112.881,165.671,59.368,160.676
C05021=1013.975,13.228,-112.894,165.672,59.359,160.675
C05022=1013.980,13.479,-112.907,165.675,59.351,160.674
C05023=1013.984,13.729,-112.920,165.676,59.342,160.672
C05024=1013.988,13.978,-112.933,165.679,59.333,160.671
C05025=1013.994,14.228,-112.947,165.682,59.325,160.671
C05026=1013.998,14.477,-112.960,165.683,59.316,160.669
C05027=1014.003,14.727,-112.972,165.686,59.308,160.668
C05028=1014.008,14.977,-112.986,165.688,59.299,160.667
C05029=1014.013,15.226,-112.998,165.689,59.290,160.666
C05030=1014.018,15.475,-113.012,165.692,59.282,160.665
C05031=1014.023,15.725,-113.025,165.694,59.273,160.664
C05032=1014.027,15.975,-113.038,165.696,59.264,160.662
C05033=1014.032,16.224,-113.051,165.699,59.256,160.662
C05034=1014.037,16.474,-113.064,165.701,59.246,160.661
C05035=1014.042,16.723,-113.077,165.703,59.237,160.659
C05036=1014.047,16.973,-113.090,165.705,59.229,160.658
C05037=1014.052,17.223,-113.103,165.707,59.220,160.657
C05038=1014.056,17.473,-113.116,165.710,59.211,160.656
C05039=1014.061,17.721,-113.129,165.712,59.202,160.655
C05040=1014.066,17.972,-113.143,165.713,59.193,160.654
C05041=1014.071,18.221,-113.155,165.716,59.184,160.652
C05042=1014.076,18.471,-113.169,165.719,59.176,160.652
C05043=1014.081,18.720,-113.182,165.721,59.167,160.650
C05044=1014.086,18.970,-113.195,165.722,59.158,160.649
C05045=1014.090,19.220,-113.209,165.725,59.149,160.648
C05046=1014.095,19.469,-113.222,165.728,59.141,160.647
C05047=1014.100,19.719,-113.235,165.730,59.132,160.646
C05048=1014.105,19.969,-113.248,165.731,59.123,160.645
C05049=1014.109,20.218,-113.262,165.733,59.114,160.644
C05050=1014.114,20.468,-113.275,165.736,59.105,160.642
C05051=1014.118,20.718,-113.288,165.738,59.096,160.641
C05052=1014.124,20.967,-113.302,165.740,59.088,160.640
C05053=1014.128,21.217,-113.315,165.742,59.079,160.639
C05054=1014.133,21.466,-113.328,165.745,59.070,160.638
C05055=1014.138,21.716,-113.342,165.747,59.061,160.637
C05056=1014.142,21.966,-113.355,165.748,59.052,160.636
C05057=1014.148,22.215,-113.369,165.751,59.043,160.634
C05058=1014.152,22.465,-113.381,165.753,59.034,160.633
C05059=1014.158,22.714,-113.395,165.755,59.025,160.632
C05060=1014.162,22.964,-113.409,165.758,59.016,160.631
C05061=1014.167,23.214,-113.422,165.760,59.007,160.630
C05062=1014.172,23.463,-113.435,165.761,58.998,160.629
C05063=1014.177,23.712,-113.449,165.764,58.989,160.627
C05064=1014.182,23.962,-113.462,165.766,58.980,160.626
C05065=1014.186,24.212,-113.475,165.768,58.971,160.625
C05066=1014.191,24.462,-113.489,165.771,58.962,160.624
C05067=1014.196,24.711,-113.502,165.773,58.953,160.623
C05068=1014.201,24.961,-113.516,165.776,58.944,160.622
C05069=1014.206,25.210,-113.529,165.778,58.935,160.621
C05070=1014.210,25.460,-113.543,165.779,58.926,160.619
C05071=1014.215,25.709,-113.556,165.782,58.917,160.618
C05072=1014.221,25.990,-113.571,165.784,58.907,160.617
C05073=1014.226,26.270,-113.587,165.787,58.896,160.616
C05074=1014.232,26.551,-113.602,165.790,58.886,160.614
C05075=1014.237,26.831,-113.617,165.792,58.876,160.613
C05076=1014.242,27.080,-113.630,165.794,58.867,160.612
C05077=1014.247,27.330,-113.644,165.796,58.858,160.610
C05078=1014.252,27.580,-113.657,165.798,58.849,160.609
C05079=1014.256,27.830,-113.672,165.801,58.839,160.608
C05080=1014.261,28.079,-113.685,165.803,58.830,160.607
C05081=1014.265,28.329,-113.699,165.805,58.822,160.606
C05082=1014.271,28.579,-113.713,165.807,58.813,160.605
C05083=1014.276,28.827,-113.726,165.809,58.804,160.603
C05084=1014.280,29.077,-113.741,165.812,58.795,160.602
C05085=1014.285,29.327,-113.753,165.814,58.786,160.601
C05086=1014.290,29.577,-113.768,165.817,58.777,160.600
C05087=1014.295,29.826,-113.781,165.819,58.768,160.599
C05088=1014.299,30.076,-113.795,165.821,58.758,160.598
C05089=1014.304,30.326,-113.809,165.823,58.749,160.596
C05090=1014.309,30.575,-113.823,165.826,58.740,160.595
C05091=1014.314,30.824,-113.837,165.827,58.731,160.594
C05092=1014.318,31.074,-113.850,165.829,58.722,160.593
C05093=1014.323,31.324,-113.864,165.831,58.712,160.591
C05094=1014.328,31.573,-113.878,165.834,58.703,160.590
C05095=1014.333,31.823,-113.892,165.836,58.694,160.589
C05096=1014.338,32.073,-113.905,165.838,58.685,160.588
C05097=1014.342,32.322,-113.919,165.841,58.676,160.587
C05098=1014.348,32.572,-113.933,165.843,58.666,160.586
C05099=1014.352,32.821,-113.947,165.845,58.657,160.584
C05100=1014.357,33.070,-113.961,165.848,58.648,160.583
C05101=1014.362,33.321,-113.975,165.849,58.639,160.582
C05102=1014.367,33.570,-113.988,165.852,58.630,160.581
C05103=1014.372,33.819,-114.002,165.854,58.621,160.580
C05104=1014.376,34.068,-114.016,165.856,58.611,160.578
C05105=1014.382,34.318,-114.030,165.858,58.602,160.577
C05106=1014.386,34.569,-114.044,165.861,58.593,160.576
C05107=1014.391,34.817,-114.057,165.863,58.583,160.575
C05108=1014.396,35.067,-114.072,165.865,58.574,160.573
C05109=1014.401,35.316,-114.085,165.867,58.564,160.572
C05110=1014.405,35.566,-114.100,165.869,58.555,160.571
C05111=1014.411,35.816,-114.114,165.872,58.546,160.570
C05112=1014.415,36.065,-114.127,165.874,58.537,160.568
C05113=1014.420,36.315,-114.141,165.876,58.527,160.567
C05114=1014.425,36.565,-114.155,165.878,58.518,160.566
C05115=1014.429,36.814,-114.170,165.881,58.509,160.565
C05116=1014.435,37.064,-114.183,165.883,58.500,160.564
C05117=1014.439,37.314,-114.198,165.885,58.490,160.562
C05118=1014.443,37.563,-114.212,165.887,58.481,160.561
C05119=1014.449,37.812,-114.226,165.890,58.472,160.560
C05120=1014.454,38.062,-114.240,165.892,58.462,160.559
C05121=1014.458,38.311,-114.254,165.894,58.453,160.557
C05122=1014.463,38.561,-114.269,165.897,58.444,160.556
C05123=1014.468,38.811,-114.283,165.899,58.435,160.555
C05124=1014.473,39.061,-114.297,165.901,58.426,160.554
C05125=1014.477,39.310,-114.311,165.903,58.416,160.552
C05126=1014.483,39.559,-114.326,165.905,58.407,160.551
C05127=1014.487,39.809,-114.340,165.907,58.397,160.550
C05128=1014.492,40.058,-114.354,165.911,58.388,160.549
C05129=1014.496,40.308,-114.369,165.913,58.379,160.548
C05130=1014.502,40.557,-114.383,165.915,58.369,160.547
C05131=1014.506,40.807,-114.397,165.918,58.360,160.545
C05132=1014.511,41.056,-114.411,165.920,58.350,160.544
C05133=1014.516,41.306,-114.425,165.922,58.341,160.543
C05134=1014.521,41.556,-114.440,165.924,58.332,160.541
C05135=1014.525,41.805,-114.454,165.926,58.322,160.540
C05136=1014.531,42.086,-114.470,165.929,58.312,160.539
C05137=1014.536,42.366,-114.486,165.931,58.301,160.537
C05138=1014.541,42.647,-114.503,165.934,58.291,160.536
C05139=1014.547,42.928,-114.519,165.937,58.280,160.535
C05140=1014.552,43.178,-114.533,165.938,58.271,160.533
C05141=1014.556,43.426,-114.548,165.940,58.262,160.532
C05142=1014.561,43.676,-114.563,165.942,58.253,160.531
C05143=1014.566,43.926,-114.577,165.945,58.244,160.530
C05144=1014.571,44.175,-114.592,165.947,58.235,160.529
C05145=1014.575,44.424,-114.606,165.949,58.225,160.527
C05146=1014.579,44.674,-114.621,165.953,58.215,160.526
C05147=1014.584,44.924,-114.635,165.955,58.206,160.525
C05148=1014.589,45.173,-114.650,165.957,58.197,160.524
C05149=1014.594,45.423,-114.665,165.959,58.187,160.522
C05150=1014.598,45.672,-114.679,165.962,58.178,160.521
C05151=1014.603,45.922,-114.694,165.964,58.168,160.520
C05152=1014.607,46.172,-114.709,165.966,58.159,160.519
C05153=1014.612,46.421,-114.724,165.968,58.150,160.517
C05154=1014.616,46.670,-114.738,165.970,58.140,160.516
C05155=1014.621,46.920,-114.753,165.973,58.131,160.515
C05156=1014.626,47.169,-114.768,165.975,58.121,160.514
C05157=1014.631,47.419,-114.782,165.977,58.113,160.513
C05158=1014.636,47.669,-114.797,165.979,58.103,160.511
C05159=1014.641,47.919,-114.812,165.982,58.094,160.510
C05160=1014.645,48.168,-114.826,165.984,58.084,160.509
C05161=1014.650,48.417,-114.841,165.987,58.074,160.507
C05162=1014.655,48.667,-114.856,165.989,58.065,160.506
C05163=1014.659,48.917,-114.870,165.991,58.055,160.505
C05164=1014.664,49.166,-114.885,165.993,58.046,160.504
C05165=1014.669,49.416,-114.900,165.996,58.037,160.502
C05166=1014.674,49.664,-114.915,165.998,58.027,160.501
C05167=1014.678,49.914,-114.929,166.000,58.017,160.500
C05168=1014.683,50.164,-114.944,166.002,58.009,160.499
C05169=1014.688,50.413,-114.959,166.005,57.998,160.497
C05170=1014.693,50.663,-114.973,166.007,57.989,160.496
C05171=1014.698,50.913,-114.988,166.009,57.979,160.495
C05172=1014.703,51.163,-115.003,166.012,57.970,160.494
C05173=1014.707,51.411,-115.018,166.014,57.960,160.492
C05174=1014.712,51.661,-115.032,166.016,57.951,160.491
C05175=1014.717,51.910,-115.047,166.019,57.941,160.490
C05176=1014.722,52.160,-115.062,166.021,57.931,160.488
C05177=1014.727,52.409,-115.077,166.024,57.922,160.487
C05178=1014.731,52.659,-115.091,166.025,57.912,160.486
C05179=1014.736,52.909,-115.107,166.027,57.903,160.484
C05180=1014.741,53.158,-115.121,166.031,57.893,160.483
C05181=1014.746,53.407,-115.136,166.033,57.883,160.482
C05182=1014.750,53.657,-115.150,166.035,57.873,160.480
C05183=1014.755,53.906,-115.166,166.037,57.864,160.479
C05184=1014.760,54.156,-115.180,166.040,57.854,160.478
C05185=1014.765,54.405,-115.195,166.042,57.845,160.477
C05186=1014.770,54.655,-115.210,166.044,57.835,160.475
C05187=1014.775,54.904,-115.225,166.046,57.825,160.474
C05188=1014.780,55.154,-115.239,166.049,57.815,160.473
C05189=1014.785,55.404,-115.254,166.051,57.806,160.471
C05190=1014.789,55.654,-115.269,166.053,57.796,160.470
C05191=1014.794,55.903,-115.284,166.057,57.786,160.469
C05192=1014.799,56.153,-115.299,166.059,57.776,160.468
C05193=1014.804,56.402,-115.314,166.061,57.767,160.466
C05194=1014.809,56.651,-115.329,166.063,57.757,160.465
C05195=1014.814,56.901,-115.343,166.066,57.747,160.464
C05196=1014.818,57.150,-115.358,166.068,57.737,160.462
C05197=1014.823,57.400,-115.373,166.070,57.728,160.461
C05198=1014.828,57.649,-115.388,166.073,57.718,160.460
C05199=1014.833,57.899,-115.402,166.075,57.708,160.458
C05200=1014.839,58.180,-115.420,166.077,57.697,160.457
C05201=1014.845,58.460,-115.437,166.080,57.686,160.455
C05202=1014.849,58.741,-115.453,166.084,57.675,160.454
C05203=1014.855,59.021,-115.470,166.086,57.664,160.453
C05204=1014.860,59.270,-115.485,166.088,57.655,160.451
C05205=1014.865,59.520,-115.499,166.091,57.644,160.450
C05206=1014.870,59.769,-115.515,166.093,57.634,160.448
C05207=1014.875,60.019,-115.529,166.095,57.625,160.447
C05208=1014.880,60.269,-115.544,166.098,57.615,160.446
C05209=1014.884,60.518,-115.560,166.100,57.605,160.444
C05210=1014.889,60.768,-115.574,166.103,57.595,160.443
C05211=1014.894,61.017,-115.590,166.105,57.586,160.442
C05212=1014.899,61.267,-115.605,166.107,57.575,160.440
C05213=1014.904,61.516,-115.619,166.110,57.565,160.439
C05214=1014.909,61.766,-115.634,166.112,57.556,160.438
C05215=1014.914,62.015,-115.650,166.115,57.545,160.437
C05216=1014.919,62.265,-115.664,166.117,57.536,160.435
C05217=1014.924,62.514,-115.679,166.119,57.526,160.434
C05218=1014.929,62.763,-115.694,166.122,57.516,160.432
C05219=1014.934,63.013,-115.710,166.124,57.506,160.431
C05220=1014.939,63.263,-115.726,166.126,57.496,160.430
C05221=1014.943,63.513,-115.740,166.129,57.486,160.429
C05222=1014.948,63.762,-115.755,166.131,57.477,160.427
C05223=1014.953,64.012,-115.771,166.133,57.467,160.426
C05224=1014.958,64.261,-115.786,166.137,57.457,160.425
C05225=1014.962,64.511,-115.802,166.139,57.447,160.423
C05226=1014.967,64.760,-115.817,166.141,57.438,160.422
C05227=1014.972,65.009,-115.832,166.144,57.428,160.421
C05228=1014.977,65.259,-115.848,166.146,57.418,160.419
C05229=1014.982,65.508,-115.863,166.148,57.409,160.418
C05230=1014.987,65.757,-115.879,166.151,57.399,160.417
C05231=1014.991,66.007,-115.894,166.154,57.389,160.416
C05232=1014.996,66.257,-115.909,166.155,57.379,160.414
C05233=1015.001,66.507,-115.925,166.158,57.369,160.413
C05234=1015.006,66.756,-115.940,166.160,57.359,160.411
C05235=1015.011,67.005,-115.955,166.163,57.350,160.410
C05236=1015.015,67.255,-115.971,166.166,57.340,160.409
C05237=1015.020,67.504,-115.986,166.168,57.330,160.408
C05238=1015.024,67.754,-116.002,166.170,57.320,160.406
C05239=1015.029,68.003,-116.017,166.173,57.310,160.405
C05240=1015.034,68.253,-116.033,166.175,57.300,160.403
C05241=1015.039,68.501,-116.049,166.177,57.291,160.402
C05242=1015.044,68.752,-116.065,166.180,57.281,160.401
C05243=1015.049,69.001,-116.080,166.182,57.271,160.400
C05244=1015.053,69.250,-116.096,166.184,57.261,160.398
C05245=1015.058,69.500,-116.111,166.188,57.251,160.397
C05246=1015.063,69.749,-116.127,166.190,57.242,160.396
C05247=1015.068,69.999,-116.142,166.192,57.232,160.394
C05248=1015.072,70.248,-116.158,166.195,57.222,160.393
C05249=1015.077,70.497,-116.173,166.197,57.212,160.392
C05250=1015.082,70.747,-116.190,166.199,57.203,160.390
C05251=1015.087,70.997,-116.206,166.202,57.193,160.389
C05252=1015.092,71.246,-116.221,166.204,57.183,160.388
C05253=1015.096,71.496,-116.237,166.207,57.173,160.386
C05254=1015.101,71.745,-116.252,166.209,57.163,160.385
C05255=1015.105,71.994,-116.267,166.211,57.153,160.384
C05256=1015.110,72.244,-116.284,166.214,57.144,160.382
C05257=1015.115,72.493,-116.300,166.217,57.134,160.381
C05258=1015.120,72.743,-116.315,166.219,57.124,160.380
C05259=1015.125,72.992,-116.330,166.221,57.114,160.378
C05260=1015.129,73.242,-116.346,166.224,57.104,160.377
C05261=1015.135,73.491,-116.362,166.226,57.094,160.376
C05262=1015.139,73.741,-116.378,166.229,57.084,160.375
C05263=1015.144,73.990,-116.394,166.231,57.074,160.373
C05264=1015.149,74.271,-116.411,166.234,57.063,160.372
C05265=1015.155,74.551,-116.430,166.237,57.052,160.370
C05266=1015.160,74.832,-116.447,166.240,57.041,160.369
C05267=1015.166,75.113,-116.465,166.242,57.030,160.367
C05268=1015.170,75.362,-116.480,166.245,57.019,160.366
C05269=1015.175,75.611,-116.497,166.247,57.010,160.364
C05270=1015.180,75.861,-116.512,166.250,57.000,160.363
C05271=1015.185,76.111,-116.528,166.252,56.990,160.362
C05272=1015.189,76.360,-116.544,166.254,56.980,160.360
C05273=1015.194,76.609,-116.560,166.258,56.970,160.359
C05274=1015.199,76.859,-116.576,166.260,56.961,160.358
C05275=1015.204,77.108,-116.592,166.263,56.950,160.356
C05276=1015.208,77.358,-116.608,166.265,56.941,160.355
C05277=1015.212,77.607,-116.624,166.267,56.931,160.354
C05278=1015.218,77.857,-116.641,166.270,56.921,160.353
C05279=1015.223,78.106,-116.656,166.273,56.912,160.351
C05280=1015.227,78.355,-116.672,166.274,56.901,160.350
C05281=1015.232,78.605,-116.688,166.278,56.891,160.349
C05282=1015.237,78.854,-116.705,166.280,56.882,160.347
C05283=1015.241,79.104,-116.721,166.282,56.872,160.346
C05284=1015.246,79.353,-116.737,166.285,56.862,160.344
C05285=1015.251,79.603,-116.753,166.287,56.852,160.343
C05286=1015.255,79.852,-116.770,166.290,56.842,160.342
C05287=1015.260,80.102,-116.786,166.293,56.833,160.341
C05288=1015.265,80.350,-116.802,166.294,56.823,160.339
C05289=1015.270,80.601,-116.818,166.298,56.813,160.338
C05290=1015.274,80.850,-116.834,166.300,56.803,160.337
C05291=1015.279,81.099,-116.850,166.303,56.793,160.335
C05292=1015.284,81.349,-116.867,166.305,56.783,160.334
C05293=1015.288,81.598,-116.883,166.307,56.774,160.333
C05294=1015.293,81.847,-116.899,166.310,56.763,160.331
C05295=1015.298,82.098,-116.915,166.312,56.753,160.330
C05296=1015.303,82.346,-116.931,166.316,56.743,160.329
C05297=1015.308,82.595,-116.948,166.317,56.733,160.327
C05298=1015.312,82.845,-116.963,166.321,56.723,160.326
C05299=1015.317,83.095,-116.980,166.323,56.714,160.325
C05300=1015.322,83.344,-116.996,166.325,56.704,160.323
C05301=1015.326,83.593,-117.013,166.328,56.694,160.322
C05302=1015.331,83.843,-117.029,166.330,56.684,160.321
C05303=1015.336,84.092,-117.045,166.333,56.674,160.319
C05304=1015.341,84.342,-117.062,166.335,56.664,160.318
C05305=1015.345,84.592,-117.078,166.338,56.654,160.316
C05306=1015.351,84.840,-117.094,166.341,56.644,160.315
C05307=1015.355,85.091,-117.110,166.343,56.633,160.314
C05308=1015.360,85.339,-117.126,166.346,56.624,160.312
C05309=1015.365,85.588,-117.143,166.349,56.614,160.311
C05310=1015.370,85.839,-117.159,166.351,56.604,160.310
C05311=1015.374,86.088,-117.175,166.354,56.594,160.309
C05312=1015.379,86.338,-117.192,166.356,56.584,160.307
C05313=1015.384,86.587,-117.208,166.359,56.574,160.306
C05314=1015.388,86.836,-117.224,166.361,56.564,160.304
C05315=1015.394,87.086,-117.240,166.364,56.554,160.303
C05316=1015.399,87.335,-117.256,166.366,56.544,160.302
C05317=1015.403,87.584,-117.273,166.370,56.534,160.300
C05318=1015.408,87.834,-117.289,166.371,56.524,160.299
C05319=1015.413,88.083,-117.306,166.375,56.514,160.298
C05320=1015.418,88.333,-117.322,166.377,56.504,160.296
C05321=1015.422,88.582,-117.338,166.379,56.493,160.295
C05322=1015.427,88.832,-117.355,166.382,56.484,160.293
C05323=1015.432,89.081,-117.372,166.385,56.474,160.292
C05324=1015.437,89.330,-117.388,166.387,56.463,160.291
C05325=1015.441,89.580,-117.405,166.390,56.454,160.290
C05326=1015.446,89.829,-117.422,166.393,56.444,160.288
C05327=1015.451,90.079,-117.438,166.396,56.434,160.287
C05328=1015.456,90.360,-117.457,166.398,56.423,160.286
C05329=1015.461,90.641,-117.476,166.401,56.412,160.284
C05330=1015.467,90.921,-117.495,166.404,56.400,160.282
C05331=1015.471,91.201,-117.514,166.407,56.389,160.281
C05332=1015.479,91.562,-117.538,166.411,56.375,160.279
C05333=1015.485,91.925,-117.562,166.415,56.361,160.277
C05334=1015.492,92.286,-117.586,166.418,56.346,160.275
C05335=1015.500,92.647,-117.610,166.422,56.332,160.273
C05336=1015.503,92.896,-117.627,166.425,56.322,160.272
C05337=1015.509,93.146,-117.644,166.427,56.312,160.270
C05338=1015.513,93.395,-117.661,166.430,56.302,160.269
C05339=1015.518,93.644,-117.678,166.432,56.292,160.268
C05340=1015.522,93.894,-117.695,166.436,56.282,160.267
C05341=1015.528,94.143,-117.711,166.438,56.272,160.265
C05342=1015.532,94.392,-117.728,166.441,56.262,160.264
C05343=1015.537,94.642,-117.745,166.443,56.252,160.262
C05344=1015.542,94.891,-117.761,166.446,56.242,160.261
C05345=1015.546,95.141,-117.779,166.448,56.232,160.260
C05346=1015.551,95.390,-117.795,166.452,56.222,160.259
C05347=1015.556,95.639,-117.812,166.454,56.212,160.257
C05348=1015.561,95.888,-117.829,166.457,56.202,160.256
C05349=1015.566,96.138,-117.845,166.459,56.192,160.254
C05350=1015.570,96.387,-117.862,166.462,56.181,160.253
C05351=1015.575,96.637,-117.879,166.465,56.171,160.252
C05352=1015.580,96.886,-117.896,166.467,56.161,160.250
C05353=1015.585,97.136,-117.913,166.471,56.152,160.249
C05354=1015.589,97.385,-117.930,166.473,56.141,160.248
C05355=1015.594,97.634,-117.947,166.475,56.131,160.246
C05356=1015.599,97.884,-117.963,166.478,56.121,160.245
C05357=1015.604,98.133,-117.980,166.481,56.111,160.244
C05358=1015.609,98.383,-117.997,166.484,56.101,160.243
C05359=1015.613,98.632,-118.014,166.486,56.091,160.241
C05360=1015.618,98.882,-118.031,166.489,56.081,160.240
C05361=1015.623,99.131,-118.047,166.492,56.071,160.238
C05362=1015.628,99.380,-118.065,166.495,56.061,160.237
C05363=1015.632,99.630,-118.083,166.497,56.051,160.236
C05364=1015.637,99.879,-118.099,166.501,56.041,160.235
C05365=1015.641,100.129,-118.117,166.502,56.031,160.233
C05366=1015.646,100.378,-118.133,166.506,56.022,160.232
C05367=1015.651,100.627,-118.151,166.508,56.011,160.230
C05368=1015.656,100.877,-118.168,166.511,56.002,160.229
C05369=1015.660,101.126,-118.185,166.513,55.992,160.228
C05370=1015.665,101.375,-118.203,166.517,55.982,160.227
C05371=1015.669,101.624,-118.220,166.519,55.972,160.225
C05372=1015.674,101.874,-118.237,166.522,55.962,160.224
C05373=1015.679,102.124,-118.254,166.524,55.952,160.222
C05374=1015.684,102.372,-118.271,166.527,55.941,160.221
C05375=1015.688,102.622,-118.289,166.530,55.932,160.220
